LIN {X 0,Y 355.805,Z 517.624,A -85,B 0,C 180,E1 -17546.603,E2 -17546.603} C_VEL
LIN {X 0,Y 356.856,Z 517.924,A -85,B 0,C 180,E1 -17547.743,E2 -17547.743} C_VEL
LIN {X 0,Y 357.535,Z 518.046,A -85,B 0,C 180,E1 -17548.874,E2 -17548.874} C_VEL
LIN {X 0,Y 357.744,Z 518.094,A -85,B 0,C 180,E1 -17550,E2 -17550} C_VEL
LIN {X 0,Y 357.534,Z 518.031,A -85,B 0,C 180,E1 -17551.127,E2 -17551.127} C_VEL
LIN {X 0,Y 356.823,Z 517.932,A -85,B 0,C 180,E1 -17552.258,E2 -17552.258} C_VEL
LIN {X 0,Y 355.806,Z 517.611,A -85,B 0,C 180,E1 -17553.397,E2 -17553.397} C_VEL
LIN {X 0,Y 354.452,Z 517.067,A -85,B 0,C 180,E1 -17554.549,E2 -17554.549} C_VEL
LIN {X 0,Y 352.887,Z 516.184,A -85,B 0,C 180,E1 -17555.715,E2 -17555.715} C_VEL
LIN {X 0,Y 351.141,Z 514.881,A -85,B 0,C 180,E1 -17556.897,E2 -17556.897} C_VEL
LIN {X 0,Y 348.325,Z 512.278,A -85,B 0,C 180,E1 -17558.645,E2 -17558.645} C_VEL
LIN {X 0,Y 346.106,Z 510.135,A -85,B 0,C 180,E1 -17559.805,E2 -17559.805} C_VEL
LIN {X 0,Y 342.78,Z 507.679,A -85,B 0,C 180,E1 -17561.152,E2 -17561.152} C_VEL
LIN {X 0,Y 338.634,Z 503.933,A -85,B 0,C 180,E1 -17562.729,E2 -17562.729} C_VEL
LIN {X 0,Y 333.72,Z 499.517,A -85,B 0,C 180,E1 -17564.367,E2 -17564.367} C_VEL
LIN {X 0,Y 327.515,Z 493.449,A -85,B 0,C 180,E1 -17566.198,E2 -17566.198} C_VEL
LIN {X 0,Y 321.238,Z 487.195,A -85,B 0,C 180,E1 -17567.836,E2 -17567.836} C_VEL
LIN {X 0,Y 314.724,Z 480.337,A -85,B 0,C 180,E1 -17569.36,E2 -17569.36} C_VEL
LIN {X 0,Y 306.811,Z 471.536,A -85,B 0,C 180,E1 -17571.025,E2 -17571.025} C_VEL
LIN {X 0,Y 297.528,Z 460.121,A -85,B 0,C 180,E1 -17572.896,E2 -17572.896} C_VEL
LIN {X 0,Y 290.607,Z 450.33,A -85,B 0,C 180,E1 -17574.276,E2 -17574.276} C_VEL
LIN {X 0,Y 285.444,Z 441.391,A -85,B 0,C 180,E1 -17575.305,E2 -17575.305} C_VEL
LIN {X 0,Y 279.385,Z 428.404,A -85,B 0,C 180,E1 -17576.454,E2 -17576.454} C_VEL
LIN {X 0,Y 277.455,Z 424.082,A -85,B 0,C 180,E1 -17576.78,E2 -17576.78} C_VEL
LIN {X 0,Y 277.336,Z 423.44,A -85,B 0,C 180,E1 -17576.813,E2 -17576.813} C_VEL
LIN {X 0,Y 277.268,Z 423.449,A -85,B 0,C 180,E1 -17580.482,E2 -17580.482} C_VEL
LIN {X 0,Y 277.251,Z 423.449,A -85,B 0,C 180,E1 -17583.895,E2 -17583.895} C_VEL
LIN {X 0,Y 277.287,Z 423.444,A -85,B 0,C 180,E1 -17587.466,E2 -17587.466} C_VEL
LIN {X 0,Y 277.262,Z 423.447,A -85,B 0,C 180,E1 -17591.227,E2 -17591.227} C_VEL
LIN {X 0,Y 277.239,Z 423.449,A -85,B 0,C 180,E1 -17595.218,E2 -17595.218} C_VEL
LIN {X 0,Y 277.221,Z 423.451,A -85,B 0,C 180,E1 -17599.512,E2 -17599.512} C_VEL
LIN {X 0,Y 277.277,Z 423.446,A -85,B 0,C 180,E1 -17602.533,E2 -17602.533} C_VEL
LIN {X 0,Y 277.251,Z 423.451,A -85,B 0,C 180,E1 -17606.106,E2 -17606.106} C_VEL
LIN {X 0,Y 277.258,Z 423.447,A -85,B 0,C 180,E1 -17609.539,E2 -17609.539} C_VEL
LIN {X 0,Y 277.356,Z 423.434,A -85,B 0,C 180,E1 -17612.865,E2 -17612.865} C_VEL
LIN {X 0,Y 277.326,Z 423.44,A -85,B 0,C 180,E1 -17616.08,E2 -17616.08} C_VEL
LIN {X 0,Y 277.342,Z 423.434,A -85,B 0,C 180,E1 -17620.767,E2 -17620.767} C_VEL
LIN {X 0,Y 277.432,Z 423.422,A -85,B 0,C 180,E1 -17625.327,E2 -17625.327} C_VEL
LIN {X 0,Y 277.504,Z 423.416,A -85,B 0,C 180,E1 -17629.789,E2 -17629.789} C_VEL
LIN {X 0,Y 277.651,Z 423.398,A -85,B 0,C 180,E1 -17632.73,E2 -17632.73} C_VEL
LIN {X 0,Y 277.819,Z 423.364,A -85,B 0,C 180,E1 -17638.551,E2 -17638.551} C_VEL
LIN {X 0,Y 277.82,Z 423.376,A -85,B 0,C 180,E1 -17641.45,E2 -17641.45} C_VEL
LIN {X 0,Y 277.652,Z 423.4,A -85,B 0,C 180,E1 -17647.272,E2 -17647.272} C_VEL
LIN {X 0,Y 277.505,Z 423.416,A -85,B 0,C 180,E1 -17650.212,E2 -17650.212} C_VEL
LIN {X 0,Y 277.434,Z 423.425,A -85,B 0,C 180,E1 -17654.675,E2 -17654.675} C_VEL
LIN {X 0,Y 277.344,Z 423.44,A -85,B 0,C 180,E1 -17659.235,E2 -17659.235} C_VEL
LIN {X 0,Y 277.318,Z 423.44,A -85,B 0,C 180,E1 -17664.171,E2 -17664.171} C_VEL
LIN {X 0,Y 277.305,Z 423.441,A -85,B 0,C 180,E1 -17666.304,E2 -17666.304} C_VEL
LIN {X 0,Y 276.642,Z 423.529,A -85,B 0,C 180,E1 -17667.516,E2 -17667.516} C_VEL
LIN {X 0,Y 273.724,Z 423.892,A -85,B 0,C 180,E1 -17669.489,E2 -17669.489} C_VEL
LIN {X 0,Y 271.291,Z 424.409,A -85,B 0,C 180,E1 -17671.09,E2 -17671.09} C_VEL
LIN {X 0,Y 270.324,Z 424.94,A -85,B 0,C 180,E1 -17672.33,E2 -17672.33} C_VEL
LIN {X 0,Y 270.288,Z 425.147,A -85,B 0,C 180,E1 -17672.748,E2 -17672.748} C_VEL
LIN {X 0,Y 270.646,Z 427.318,A -85,B 0,C 180,E1 -17676.674,E2 -17676.674} C_VEL
LIN {X 0,Y 271.072,Z 430.164,A -85,B 0,C 180,E1 -17681.247,E2 -17681.247} C_VEL
LIN {X 0,Y 271.313,Z 432.313,A -85,B 0,C 180,E1 -17684.38,E2 -17684.38} C_VEL
LIN {X 0,Y 271.394,Z 434.753,A -85,B 0,C 180,E1 -17687.678,E2 -17687.678} C_VEL
LIN {X 0,Y 271.049,Z 437.477,A -85,B 0,C 180,E1 -17691.067,E2 -17691.067} C_VEL
LIN {X 0,Y 270.38,Z 440.968,A -85,B 0,C 180,E1 -17695.121,E2 -17695.121} C_VEL
LIN {X 0,Y 269.721,Z 444.717,A -85,B 0,C 180,E1 -17699.303,E2 -17699.303} C_VEL
LIN {X 0,Y 269.252,Z 447.838,A -85,B 0,C 180,E1 -17702.648,E2 -17702.648} C_VEL
LIN {X 0,Y 270.086,Z 451.047,A -85,B 0,C 180,E1 -17702.876,E2 -17702.876} C_VEL
LIN {X 0,Y 273.605,Z 464.4,A -85,B 0,C 180,E1 -17704.033,E2 -17704.033} C_VEL
LIN {X 0,Y 275.695,Z 474.898,A -85,B 0,C 180,E1 -17705.107,E2 -17705.107} C_VEL
LIN {X 0,Y 276.978,Z 485.03,A -85,B 0,C 180,E1 -17706.287,E2 -17706.287} C_VEL
LIN {X 0,Y 277.683,Z 494.384,A -85,B 0,C 180,E1 -17707.542,E2 -17707.542} C_VEL
LIN {X 0,Y 277.693,Z 499.477,A -85,B 0,C 180,E1 -17708.276,E2 -17708.276} C_VEL
LIN {X 0,Y 275.78,Z 509.625,A -85,B 0,C 180,E1 -17709.877,E2 -17709.877} C_VEL
LIN {X 0,Y 274.264,Z 517.761,A -85,B 0,C 180,E1 -17711.466,E2 -17711.466} C_VEL
LIN {X 0,Y 272.829,Z 524.973,A -85,B 0,C 180,E1 -17713.154,E2 -17713.154} C_VEL
LIN {X 0,Y 271.488,Z 531.513,A -85,B 0,C 180,E1 -17714.997,E2 -17714.997} C_VEL
LIN {X 0,Y 270.522,Z 536.015,A -85,B 0,C 180,E1 -17716.478,E2 -17716.478} C_VEL
LIN {X 0,Y 269.51,Z 541.512,A -85,B 0,C 180,E1 -17718.721,E2 -17718.721} C_VEL
LIN {X 0,Y 268.783,Z 545.842,A -85,B 0,C 180,E1 -17720.974,E2 -17720.974} C_VEL
LIN {X 0,Y 268.481,Z 548.213,A -85,B 0,C 180,E1 -17722.479,E2 -17722.479} C_VEL
LIN {X 0,Y 268.216,Z 550.778,A -85,B 0,C 180,E1 -17724.695,E2 -17724.695} C_VEL
LIN {X 0,Y 268.174,Z 552.47,A -85,B 0,C 180,E1 -17726.995,E2 -17726.995} C_VEL
LIN {X 0,Y 268.18,Z 553.061,A -85,B 0,C 180,E1 -17728.498,E2 -17728.498} C_VEL
LIN {X 0,Y 268.18,Z 553.061,A -85,B 0,C 180,E1 -17731.501,E2 -17731.501} C_VEL
LIN {X 0,Y 268.174,Z 552.47,A -85,B 0,C 180,E1 -17733.004,E2 -17733.004} C_VEL
LIN {X 0,Y 268.303,Z 550.017,A -85,B 0,C 180,E1 -17736.014,E2 -17736.014} C_VEL
LIN {X 0,Y 268.619,Z 547.062,A -85,B 0,C 180,E1 -17738.273,E2 -17738.273} C_VEL
LIN {X 0,Y 269.245,Z 543.069,A -85,B 0,C 180,E1 -17740.528,E2 -17740.528} C_VEL
LIN {X 0,Y 270.139,Z 537.934,A -85,B 0,C 180,E1 -17742.775,E2 -17742.775} C_VEL
LIN {X 0,Y 271.225,Z 532.67,A -85,B 0,C 180,E1 -17744.633,E2 -17744.633} C_VEL
LIN {X 0,Y 272.503,Z 526.351,A -85,B 0,C 180,E1 -17746.48,E2 -17746.48} C_VEL
LIN {X 0,Y 274.014,Z 519.292,A -85,B 0,C 180,E1 -17748.188,E2 -17748.188} C_VEL
LIN {X 0,Y 275.03,Z 513.468,A -85,B 0,C 180,E1 -17749.402,E2 -17749.402} C_VEL
LIN {X 0,Y 276.596,Z 505.288,A -85,B 0,C 180,E1 -17750.837,E2 -17750.837} C_VEL
LIN {X 0,Y 277.891,Z 498.129,A -85,B 0,C 180,E1 -17751.902,E2 -17751.902} C_VEL
LIN {X 0,Y 277.357,Z 488.828,A -85,B 0,C 180,E1 -17753.222,E2 -17753.222} C_VEL
LIN {X 0,Y 276.224,Z 478.64,A -85,B 0,C 180,E1 -17754.473,E2 -17754.473} C_VEL
LIN {X 0,Y 274.544,Z 468.766,A -85,B 0,C 180,E1 -17755.53,E2 -17755.53} C_VEL
LIN {X 0,Y 272.201,Z 458.808,A -85,B 0,C 180,E1 -17756.472,E2 -17756.472} C_VEL
LIN {X 0,Y 269.316,Z 448.595,A -85,B 0,C 180,E1 -17757.303,E2 -17757.303} C_VEL
LIN {X 0,Y 269.25,Z 447.839,A -85,B 0,C 180,E1 -17757.351,E2 -17757.351} C_VEL
LIN {X 0,Y 269.771,Z 444.07,A -85,B 0,C 180,E1 -17761.401,E2 -17761.401} C_VEL
LIN {X 0,Y 270.366,Z 440.938,A -85,B 0,C 180,E1 -17764.88,E2 -17764.88} C_VEL
LIN {X 0,Y 271.046,Z 437.457,A -85,B 0,C 180,E1 -17768.932,E2 -17768.932} C_VEL
LIN {X 0,Y 271.389,Z 434.743,A -85,B 0,C 180,E1 -17772.322,E2 -17772.322} C_VEL
LIN {X 0,Y 271.307,Z 432.301,A -85,B 0,C 180,E1 -17775.619,E2 -17775.619} C_VEL
LIN {X 0,Y 270.971,Z 429.623,A -85,B 0,C 180,E1 -17779.577,E2 -17779.577} C_VEL
LIN {X 0,Y 270.606,Z 427.143,A -85,B 0,C 180,E1 -17783.619,E2 -17783.619} C_VEL
LIN {X 0,Y 270.333,Z 425.32,A -85,B 0,C 180,E1 -17786.91,E2 -17786.91} C_VEL
LIN {X 0,Y 270.202,Z 424.328,A -85,B 0,C 180,E1 -17789.128,E2 -17789.128} C_VEL
LIN {X 0,Y 270.263,Z 424.321,A -85,B 0,C 180,E1 -17792.144,E2 -17792.144} C_VEL
LIN {X 0,Y 270.275,Z 424.321,A -85,B 0,C 180,E1 -17795.518,E2 -17795.518} C_VEL
LIN {X 0,Y 270.298,Z 424.318,A -85,B 0,C 180,E1 -17800.243,E2 -17800.243} C_VEL
LIN {X 0,Y 270.399,Z 424.303,A -85,B 0,C 180,E1 -17804.934,E2 -17804.934} C_VEL
LIN {X 0,Y 270.438,Z 424.296,A -85,B 0,C 180,E1 -17809.518,E2 -17809.518} C_VEL
LIN {X 0,Y 270.607,Z 424.279,A -85,B 0,C 180,E1 -17812.538,E2 -17812.538} C_VEL
LIN {X 0,Y 270.783,Z 424.253,A -85,B 0,C 180,E1 -17818.512,E2 -17818.512} C_VEL
LIN {X 0,Y 270.782,Z 424.24,A -85,B 0,C 180,E1 -17821.486,E2 -17821.486} C_VEL
LIN {X 0,Y 270.606,Z 424.275,A -85,B 0,C 180,E1 -17827.46,E2 -17827.46} C_VEL
LIN {X 0,Y 270.436,Z 424.298,A -85,B 0,C 180,E1 -17830.48,E2 -17830.48} C_VEL
LIN {X 0,Y 270.397,Z 424.297,A -85,B 0,C 180,E1 -17835.064,E2 -17835.064} C_VEL
LIN {X 0,Y 270.296,Z 424.314,A -85,B 0,C 180,E1 -17839.755,E2 -17839.755} C_VEL
LIN {X 0,Y 270.268,Z 424.314,A -85,B 0,C 180,E1 -17844.585,E2 -17844.585} C_VEL
LIN {X 0,Y 270.265,Z 424.322,A -85,B 0,C 180,E1 -17847.908,E2 -17847.908} C_VEL
LIN {X 0,Y 270.179,Z 424.329,A -85,B 0,C 180,E1 -17851.348,E2 -17851.348} C_VEL
LIN {X 0,Y 270.21,Z 424.325,A -85,B 0,C 180,E1 -17854.903,E2 -17854.903} C_VEL
LIN {X 0,Y 270.216,Z 424.324,A -85,B 0,C 180,E1 -17858.717,E2 -17858.717} C_VEL
LIN {X 0,Y 270.226,Z 424.322,A -85,B 0,C 180,E1 -17862.547,E2 -17862.547} C_VEL
LIN {X 0,Y 270.23,Z 424.322,A -85,B 0,C 180,E1 -17866.735,E2 -17866.735} C_VEL
LIN {X 0,Y 270.245,Z 424.323,A -85,B 0,C 180,E1 -17869.448,E2 -17869.448} C_VEL
LIN {X 0,Y 270.252,Z 424.323,A -85,B 0,C 180,E1 -17873.721,E2 -17873.721} C_VEL
LIN {X 0,Y 270.199,Z 424.328,A -85,B 0,C 180,E1 -17876.893,E2 -17876.893} C_VEL
LIN {X 0,Y 270.224,Z 424.324,A -85,B 0,C 180,E1 -17880.387,E2 -17880.387} C_VEL
LIN {X 0,Y 270.292,Z 424.316,A -85,B 0,C 180,E1 -17882.436,E2 -17882.436} C_VEL
LIN {X 0,Y 271.238,Z 427.034,A -85,B 0,C 180,E1 -17882.635,E2 -17882.635} C_VEL
LIN {X 0,Y 277.009,Z 439.136,A -85,B 0,C 180,E1 -17883.726,E2 -17883.726} C_VEL
LIN {X 0,Y 281.643,Z 449.005,A -85,B 0,C 180,E1 -17884.788,E2 -17884.788} C_VEL
LIN {X 0,Y 287.444,Z 458.206,A -85,B 0,C 180,E1 -17886.055,E2 -17886.055} C_VEL
LIN {X 0,Y 294.179,Z 467.421,A -85,B 0,C 180,E1 -17887.528,E2 -17887.528} C_VEL
LIN {X 0,Y 304.319,Z 479.414,A -85,B 0,C 180,E1 -17889.733,E2 -17889.733} C_VEL
LIN {X 0,Y 312.848,Z 488.67,A -85,B 0,C 180,E1 -17891.67,E2 -17891.67} C_VEL
LIN {X 0,Y 318.244,Z 494.216,A -85,B 0,C 180,E1 -17893.006,E2 -17893.006} C_VEL
LIN {X 0,Y 324.415,Z 500.118,A -85,B 0,C 180,E1 -17894.656,E2 -17894.656} C_VEL
LIN {X 0,Y 330.188,Z 505.543,A -85,B 0,C 180,E1 -17896.46,E2 -17896.46} C_VEL
LIN {X 0,Y 334.168,Z 509.334,A -85,B 0,C 180,E1 -17897.86,E2 -17897.86} C_VEL
LIN {X 0,Y 338.789,Z 513.066,A -85,B 0,C 180,E1 -17899.618,E2 -17899.618} C_VEL
LIN {X 0,Y 341.625,Z 515.391,A -85,B 0,C 180,E1 -17900.914,E2 -17900.914} C_VEL
LIN {X 0,Y 345.072,Z 518.684,A -85,B 0,C 180,E1 -17902.981,E2 -17902.981} C_VEL
LIN {X 0,Y 346.856,Z 520.059,A -85,B 0,C 180,E1 -17904.186,E2 -17904.186} C_VEL
LIN {X 0,Y 348.468,Z 521.018,A -85,B 0,C 180,E1 -17905.373,E2 -17905.373} C_VEL
LIN {X 0,Y 349.853,Z 521.619,A -85,B 0,C 180,E1 -17906.545,E2 -17906.545} C_VEL
LIN {X 0,Y 350.949,Z 521.964,A -85,B 0,C 180,E1 -17907.705,E2 -17907.705} C_VEL
LIN {X 0,Y 351.691,Z 522.116,A -85,B 0,C 180,E1 -17908.855,E2 -17908.855} C_VEL
LIN {X 0,Y 351.927,Z 522.169,A -85,B 0,C 180,E1 -17910,E2 -17910} C_VEL
LIN {X 0,Y 351.503,Z 522.091,A -85,B 0,C 180,E1 -17911.422,E2 -17911.422} C_VEL
LIN {X 0,Y 350.926,Z 521.964,A -85,B 0,C 180,E1 -17912.296,E2 -17912.296} C_VEL
LIN {X 0,Y 349.852,Z 521.61,A -85,B 0,C 180,E1 -17913.455,E2 -17913.455} C_VEL
LIN {X 0,Y 348.46,Z 521.034,A -85,B 0,C 180,E1 -17914.628,E2 -17914.628} C_VEL
LIN {X 0,Y 346.357,Z 519.728,A -85,B 0,C 180,E1 -17916.145,E2 -17916.145} C_VEL
LIN {X 0,Y 343.074,Z 516.885,A -85,B 0,C 180,E1 -17918.245,E2 -17918.245} C_VEL
LIN {X 0,Y 340.788,Z 514.63,A -85,B 0,C 180,E1 -17919.496,E2 -17919.496} C_VEL
LIN {X 0,Y 336.689,Z 511.512,A -85,B 0,C 180,E1 -17921.17,E2 -17921.17} C_VEL
LIN {X 0,Y 333.433,Z 508.537,A -85,B 0,C 180,E1 -17922.427,E2 -17922.427} C_VEL
LIN {X 0,Y 328.737,Z 504.298,A -85,B 0,C 180,E1 -17924.004,E2 -17924.004} C_VEL
LIN {X 0,Y 323.411,Z 499.102,A -85,B 0,C 180,E1 -17925.642,E2 -17925.642} C_VEL
LIN {X 0,Y 318.25,Z 494.227,A -85,B 0,C 180,E1 -17927,E2 -17927} C_VEL
LIN {X 0,Y 312.849,Z 488.679,A -85,B 0,C 180,E1 -17928.331,E2 -17928.331} C_VEL
LIN {X 0,Y 302.712,Z 477.5,A -85,B 0,C 180,E1 -17930.628,E2 -17930.628} C_VEL
LIN {X 0,Y 294.181,Z 467.415,A -85,B 0,C 180,E1 -17932.473,E2 -17932.473} C_VEL
LIN {X 0,Y 286.462,Z 456.866,A -85,B 0,C 180,E1 -17934.153,E2 -17934.153} C_VEL
LIN {X 0,Y 280.871,Z 447.401,A -85,B 0,C 180,E1 -17935.397,E2 -17935.397} C_VEL
LIN {X 0,Y 276.355,Z 437.594,A -85,B 0,C 180,E1 -17936.413,E2 -17936.413} C_VEL
LIN {X 0,Y 270.48,Z 425.259,A -85,B 0,C 180,E1 -17937.501,E2 -17937.501} C_VEL
LIN {X 0,Y 270.282,Z 424.318,A -85,B 0,C 180,E1 -17937.594,E2 -17937.594} C_VEL
LIN {X 0,Y 270.181,Z 424.329,A -85,B 0,C 180,E1 -17941.348,E2 -17941.348} C_VEL
LIN {X 0,Y 270.212,Z 424.327,A -85,B 0,C 180,E1 -17944.904,E2 -17944.904} C_VEL
LIN {X 0,Y 270.219,Z 424.326,A -85,B 0,C 180,E1 -17948.717,E2 -17948.717} C_VEL
LIN {X 0,Y 270.219,Z 424.326,A -85,B 0,C 180,E1 -17952.549,E2 -17952.549} C_VEL
LIN {X 0,Y 270.185,Z 424.328,A -85,B 0,C 180,E1 -17956.746,E2 -17956.746} C_VEL
LIN {X 0,Y 270.203,Z 424.325,A -85,B 0,C 180,E1 -17961.375,E2 -17961.375} C_VEL
LIN {X 0,Y 270.22,Z 424.323,A -85,B 0,C 180,E1 -17965.098,E2 -17965.098} C_VEL
LIN {X 0,Y 270.197,Z 424.326,A -85,B 0,C 180,E1 -17969.131,E2 -17969.131} C_VEL
LIN {X 0,Y 270.261,Z 424.322,A -85,B 0,C 180,E1 -17972.147,E2 -17972.147} C_VEL
LIN {X 0,Y 270.274,Z 424.313,A -85,B 0,C 180,E1 -17975.52,E2 -17975.52} C_VEL
LIN {X 0,Y 270.299,Z 424.313,A -85,B 0,C 180,E1 -17980.245,E2 -17980.245} C_VEL
LIN {X 0,Y 270.4,Z 424.297,A -85,B 0,C 180,E1 -17984.936,E2 -17984.936} C_VEL
LIN {X 0,Y 270.439,Z 424.297,A -85,B 0,C 180,E1 -17989.52,E2 -17989.52} C_VEL
LIN {X 0,Y 270.609,Z 424.275,A -85,B 0,C 180,E1 -17992.54,E2 -17992.54} C_VEL
LIN {X 0,Y 270.785,Z 424.239,A -85,B 0,C 180,E1 -17998.514,E2 -17998.514} C_VEL
LIN {X 0,Y 270.785,Z 424.252,A -85,B 0,C 180,E1 -18001.488,E2 -18001.488} C_VEL
LIN {X 0,Y 270.61,Z 424.279,A -85,B 0,C 180,E1 -18007.462,E2 -18007.462} C_VEL
LIN {X 0,Y 270.441,Z 424.296,A -85,B 0,C 180,E1 -18010.482,E2 -18010.482} C_VEL
LIN {X 0,Y 270.402,Z 424.303,A -85,B 0,C 180,E1 -18015.065,E2 -18015.065} C_VEL
LIN {X 0,Y 270.301,Z 424.315,A -85,B 0,C 180,E1 -18019.756,E2 -18019.756} C_VEL
LIN {X 0,Y 270.274,Z 424.319,A -85,B 0,C 180,E1 -18024.586,E2 -18024.586} C_VEL
LIN {X 0,Y 270.27,Z 424.32,A -85,B 0,C 180,E1 -18027.91,E2 -18027.91} C_VEL
LIN {X 0,Y 270.195,Z 424.428,A -85,B 0,C 180,E1 -18031.348,E2 -18031.348} C_VEL
LIN {X 0,Y 270.288,Z 425.147,A -85,B 0,C 180,E1 -18032.748,E2 -18032.748} C_VEL
LIN {X 0,Y 269.753,Z 425.906,A -85,B 0,C 180,E1 -18033.985,E2 -18033.985} C_VEL
LIN {X 0,Y 267.044,Z 427.473,A -85,B 0,C 180,E1 -18035.995,E2 -18035.995} C_VEL
LIN {X 0,Y 264.743,Z 428.786,A -85,B 0,C 180,E1 -18037.628,E2 -18037.628} C_VEL
LIN {X 0,Y 263.843,Z 429.689,A -85,B 0,C 180,E1 -18038.894,E2 -18038.894} C_VEL
LIN {X 0,Y 263.82,Z 429.959,A -85,B 0,C 180,E1 -18039.322,E2 -18039.322} C_VEL
LIN {X 0,Y 264.099,Z 431.534,A -85,B 0,C 180,E1 -18041.831,E2 -18041.831} C_VEL
LIN {X 0,Y 264.332,Z 434.311,A -85,B 0,C 180,E1 -18045.88,E2 -18045.88} C_VEL
LIN {X 0,Y 264.316,Z 436.143,A -85,B 0,C 180,E1 -18048.338,E2 -18048.338} C_VEL
LIN {X 0,Y 263.778,Z 439.258,A -85,B 0,C 180,E1 -18052.208,E2 -18052.208} C_VEL
LIN {X 0,Y 263.187,Z 442.329,A -85,B 0,C 180,E1 -18055.891,E2 -18055.891} C_VEL
LIN {X 0,Y 262.626,Z 445.456,A -85,B 0,C 180,E1 -18059.44,E2 -18059.44} C_VEL
LIN {X 0,Y 262.223,Z 447.643,A -85,B 0,C 180,E1 -18061.859,E2 -18061.859} C_VEL
LIN {X 0,Y 263.126,Z 450.954,A -85,B 0,C 180,E1 -18062.103,E2 -18062.103} C_VEL
LIN {X 0,Y 266.715,Z 464.224,A -85,B 0,C 180,E1 -18063.314,E2 -18063.314} C_VEL
LIN {X 0,Y 268.981,Z 475.669,A -85,B 0,C 180,E1 -18064.543,E2 -18064.543} C_VEL
LIN {X 0,Y 270.26,Z 485.569,A -85,B 0,C 180,E1 -18065.754,E2 -18065.754} C_VEL
LIN {X 0,Y 270.914,Z 495.182,A -85,B 0,C 180,E1 -18067.1,E2 -18067.1} C_VEL
LIN {X 0,Y 270.857,Z 500.526,A -85,B 0,C 180,E1 -18067.899,E2 -18067.899} C_VEL
LIN {X 0,Y 269.123,Z 509.414,A -85,B 0,C 180,E1 -18069.357,E2 -18069.357} C_VEL
LIN {X 0,Y 267.339,Z 518.322,A -85,B 0,C 180,E1 -18071.157,E2 -18071.157} C_VEL
LIN {X 0,Y 266.03,Z 524.761,A -85,B 0,C 180,E1 -18072.71,E2 -18072.71} C_VEL
LIN {X 0,Y 264.624,Z 531.301,A -85,B 0,C 180,E1 -18074.598,E2 -18074.598} C_VEL
LIN {X 0,Y 263.603,Z 535.803,A -85,B 0,C 180,E1 -18076.116,E2 -18076.116} C_VEL
LIN {X 0,Y 262.515,Z 541.3,A -85,B 0,C 180,E1 -18078.417,E2 -18078.417} C_VEL
LIN {X 0,Y 261.752,Z 545.63,A -85,B 0,C 180,E1 -18080.729,E2 -18080.729} C_VEL
LIN {X 0,Y 261.407,Z 548,A -85,B 0,C 180,E1 -18082.274,E2 -18082.274} C_VEL
LIN {X 0,Y 261.126,Z 550.735,A -85,B 0,C 180,E1 -18084.769,E2 -18084.769} C_VEL
LIN {X 0,Y 261.09,Z 552.258,A -85,B 0,C 180,E1 -18086.914,E2 -18086.914} C_VEL
LIN {X 0,Y 261.109,Z 552.85,A -85,B 0,C 180,E1 -18088.457,E2 -18088.457} C_VEL
LIN {X 0,Y 261.109,Z 552.851,A -85,B 0,C 180,E1 -18091.542,E2 -18091.542} C_VEL
LIN {X 0,Y 261.09,Z 552.259,A -85,B 0,C 180,E1 -18093.086,E2 -18093.086} C_VEL
LIN {X 0,Y 261.233,Z 549.805,A -85,B 0,C 180,E1 -18096.177,E2 -18096.177} C_VEL
LIN {X 0,Y 261.571,Z 546.85,A -85,B 0,C 180,E1 -18098.498,E2 -18098.498} C_VEL
LIN {X 0,Y 262.238,Z 542.857,A -85,B 0,C 180,E1 -18100.812,E2 -18100.812} C_VEL
LIN {X 0,Y 263.188,Z 537.722,A -85,B 0,C 180,E1 -18103.119,E2 -18103.119} C_VEL
LIN {X 0,Y 264.332,Z 532.458,A -85,B 0,C 180,E1 -18105.024,E2 -18105.024} C_VEL
LIN {X 0,Y 265.68,Z 526.139,A -85,B 0,C 180,E1 -18106.916,E2 -18106.916} C_VEL
LIN {X 0,Y 267.022,Z 520.188,A -85,B 0,C 180,E1 -18108.411,E2 -18108.411} C_VEL
LIN {X 0,Y 268.32,Z 513.256,A -85,B 0,C 180,E1 -18109.907,E2 -18109.907} C_VEL
LIN {X 0,Y 269.931,Z 505.076,A -85,B 0,C 180,E1 -18111.377,E2 -18111.377} C_VEL
LIN {X 0,Y 271.092,Z 499.27,A -85,B 0,C 180,E1 -18112.28,E2 -18112.28} C_VEL
LIN {X 0,Y 270.601,Z 489.407,A -85,B 0,C 180,E1 -18113.738,E2 -18113.738} C_VEL
LIN {X 0,Y 269.46,Z 478.85,A -85,B 0,C 180,E1 -18115.085,E2 -18115.085} C_VEL
LIN {X 0,Y 267.765,Z 468.955,A -85,B 0,C 180,E1 -18116.192,E2 -18116.192} C_VEL
LIN {X 0,Y 265.272,Z 458.49,A -85,B 0,C 180,E1 -18117.225,E2 -18117.225} C_VEL
LIN {X 0,Y 262.348,Z 448.706,A -85,B 0,C 180,E1 -18118.078,E2 -18118.078} C_VEL
LIN {X 0,Y 262.223,Z 447.612,A -85,B 0,C 180,E1 -18118.176,E2 -18118.176} C_VEL
LIN {X 0,Y 262.685,Z 444.949,A -85,B 0,C 180,E1 -18121.112,E2 -18121.112} C_VEL
LIN {X 0,Y 263.152,Z 442.304,A -85,B 0,C 180,E1 -18124.113,E2 -18124.113} C_VEL
LIN {X 0,Y 263.771,Z 439.175,A -85,B 0,C 180,E1 -18127.793,E2 -18127.793} C_VEL
LIN {X 0,Y 264.309,Z 436.115,A -85,B 0,C 180,E1 -18131.662,E2 -18131.662} C_VEL
LIN {X 0,Y 264.333,Z 434.309,A -85,B 0,C 180,E1 -18134.12,E2 -18134.12} C_VEL
LIN {X 0,Y 264.064,Z 431.455,A -85,B 0,C 180,E1 -18138.288,E2 -18138.288} C_VEL
LIN {X 0,Y 263.666,Z 429.049,A -85,B 0,C 180,E1 -18142.188,E2 -18142.188} C_VEL
LIN {X 0,Y 263.402,Z 426.948,A -85,B 0,C 180,E1 -18145.922,E2 -18145.922} C_VEL
LIN {X 0,Y 263.151,Z 425.206,A -85,B 0,C 180,E1 -18149.506,E2 -18149.506} C_VEL
LIN {X 0,Y 263.191,Z 425.205,A -85,B 0,C 180,E1 -18153.002,E2 -18153.002} C_VEL
LIN {X 0,Y 263.182,Z 425.206,A -85,B 0,C 180,E1 -18156.386,E2 -18156.386} C_VEL
LIN {X 0,Y 263.261,Z 425.193,A -85,B 0,C 180,E1 -18159.692,E2 -18159.692} C_VEL
LIN {X 0,Y 263.347,Z 425.183,A -85,B 0,C 180,E1 -18164.521,E2 -18164.521} C_VEL
LIN {X 0,Y 263.37,Z 425.177,A -85,B 0,C 180,E1 -18169.233,E2 -18169.233} C_VEL
LIN {X 0,Y 263.569,Z 425.155,A -85,B 0,C 180,E1 -18172.337,E2 -18172.337} C_VEL
LIN {X 0,Y 263.747,Z 425.129,A -85,B 0,C 180,E1 -18178.472,E2 -18178.472} C_VEL
LIN {X 0,Y 263.747,Z 425.115,A -85,B 0,C 180,E1 -18181.526,E2 -18181.526} C_VEL
LIN {X 0,Y 263.567,Z 425.153,A -85,B 0,C 180,E1 -18187.661,E2 -18187.661} C_VEL
LIN {X 0,Y 263.368,Z 425.177,A -85,B 0,C 180,E1 -18190.765,E2 -18190.765} C_VEL
LIN {X 0,Y 263.345,Z 425.176,A -85,B 0,C 180,E1 -18195.477,E2 -18195.477} C_VEL
LIN {X 0,Y 263.258,Z 425.19,A -85,B 0,C 180,E1 -18200.306,E2 -18200.306} C_VEL
LIN {X 0,Y 263.203,Z 425.193,A -85,B 0,C 180,E1 -18205.291,E2 -18205.291} C_VEL
LIN {X 0,Y 263.17,Z 425.201,A -85,B 0,C 180,E1 -18208.73,E2 -18208.73} C_VEL
LIN {X 0,Y 263.128,Z 425.208,A -85,B 0,C 180,E1 -18212.288,E2 -18212.288} C_VEL
LIN {X 0,Y 263.185,Z 425.202,A -85,B 0,C 180,E1 -18215.977,E2 -18215.977} C_VEL
LIN {X 0,Y 263.155,Z 425.206,A -85,B 0,C 180,E1 -18219.862,E2 -18219.862} C_VEL
LIN {X 0,Y 263.186,Z 425.202,A -85,B 0,C 180,E1 -18223.97,E2 -18223.97} C_VEL
LIN {X 0,Y 263.209,Z 425.198,A -85,B 0,C 180,E1 -18228.384,E2 -18228.384} C_VEL
LIN {X 0,Y 263.201,Z 425.201,A -85,B 0,C 180,E1 -18233.23,E2 -18233.23} C_VEL
LIN {X 0,Y 263.179,Z 425.203,A -85,B 0,C 180,E1 -18235.891,E2 -18235.891} C_VEL
LIN {X 0,Y 263.146,Z 425.208,A -85,B 0,C 180,E1 -18239.507,E2 -18239.507} C_VEL
LIN {X 0,Y 263.239,Z 425.356,A -85,B 0,C 180,E1 -18241.671,E2 -18241.671} C_VEL
LIN {X 0,Y 264.24,Z 428.061,A -85,B 0,C 180,E1 -18241.871,E2 -18241.871} C_VEL
LIN {X 0,Y 270.073,Z 439.995,A -85,B 0,C 180,E1 -18243.032,E2 -18243.032} C_VEL
LIN {X 0,Y 274.341,Z 449.708,A -85,B 0,C 180,E1 -18244.1,E2 -18244.1} C_VEL
LIN {X 0,Y 279.36,Z 458.841,A -85,B 0,C 180,E1 -18245.35,E2 -18245.35} C_VEL
LIN {X 0,Y 286.308,Z 468.777,A -85,B 0,C 180,E1 -18246.997,E2 -18246.997} C_VEL
LIN {X 0,Y 295.215,Z 479.692,A -85,B 0,C 180,E1 -18249.079,E2 -18249.079} C_VEL
LIN {X 0,Y 304.329,Z 489.654,A -85,B 0,C 180,E1 -18251.23,E2 -18251.23} C_VEL
LIN {X 0,Y 311.289,Z 496.914,A -85,B 0,C 180,E1 -18252.933,E2 -18252.933} C_VEL
LIN {X 0,Y 317.614,Z 503.043,A -85,B 0,C 180,E1 -18254.602,E2 -18254.602} C_VEL
LIN {X 0,Y 322.651,Z 507.913,A -85,B 0,C 180,E1 -18256.137,E2 -18256.137} C_VEL
LIN {X 0,Y 326.992,Z 511.865,A -85,B 0,C 180,E1 -18257.589,E2 -18257.589} C_VEL
LIN {X 0,Y 330.678,Z 515.161,A -85,B 0,C 180,E1 -18258.973,E2 -18258.973} C_VEL
LIN {X 0,Y 334.773,Z 518.27,A -85,B 0,C 180,E1 -18260.636,E2 -18260.636} C_VEL
LIN {X 0,Y 336.545,Z 519.984,A -85,B 0,C 180,E1 -18261.595,E2 -18261.595} C_VEL
LIN {X 0,Y 339.546,Z 522.728,A -85,B 0,C 180,E1 -18263.464,E2 -18263.464} C_VEL
LIN {X 0,Y 342.109,Z 524.43,A -85,B 0,C 180,E1 -18265.287,E2 -18265.287} C_VEL
LIN {X 0,Y 343.57,Z 525.106,A -85,B 0,C 180,E1 -18266.482,E2 -18266.482} C_VEL
LIN {X 0,Y 344.733,Z 525.526,A -85,B 0,C 180,E1 -18267.663,E2 -18267.663} C_VEL
LIN {X 0,Y 345.535,Z 525.727,A -85,B 0,C 180,E1 -18268.835,E2 -18268.835} C_VEL
LIN {X 0,Y 345.825,Z 525.776,A -85,B 0,C 180,E1 -18270,E2 -18270} C_VEL
LIN {X 0,Y 345.532,Z 525.715,A -85,B 0,C 180,E1 -18271.166,E2 -18271.166} C_VEL
LIN {X 0,Y 344.669,Z 525.505,A -85,B 0,C 180,E1 -18272.397,E2 -18272.397} C_VEL
LIN {X 0,Y 343.568,Z 525.105,A -85,B 0,C 180,E1 -18273.519,E2 -18273.519} C_VEL
LIN {X 0,Y 342.105,Z 524.449,A -85,B 0,C 180,E1 -18274.714,E2 -18274.714} C_VEL
LIN {X 0,Y 339.546,Z 522.749,A -85,B 0,C 180,E1 -18276.536,E2 -18276.536} C_VEL
LIN {X 0,Y 336.541,Z 520.012,A -85,B 0,C 180,E1 -18278.406,E2 -18278.406} C_VEL
LIN {X 0,Y 333.971,Z 517.673,A -85,B 0,C 180,E1 -18279.692,E2 -18279.692} C_VEL
LIN {X 0,Y 328.891,Z 513.6,A -85,B 0,C 180,E1 -18281.712,E2 -18281.712} C_VEL
LIN {X 0,Y 324.818,Z 509.797,A -85,B 0,C 180,E1 -18283.185,E2 -18283.185} C_VEL
LIN {X 0,Y 319.774,Z 505.182,A -85,B 0,C 180,E1 -18284.756,E2 -18284.756} C_VEL
LIN {X 0,Y 314.681,Z 500.242,A -85,B 0,C 180,E1 -18286.191,E2 -18286.191} C_VEL
LIN {X 0,Y 308.211,Z 493.741,A -85,B 0,C 180,E1 -18287.826,E2 -18287.826} C_VEL
LIN {X 0,Y 300.492,Z 485.615,A -85,B 0,C 180,E1 -18289.665,E2 -18289.665} C_VEL
LIN {X 0,Y 291.511,Z 475.332,A -85,B 0,C 180,E1 -18291.789,E2 -18291.789} C_VEL
LIN {X 0,Y 283.765,Z 465.367,A -85,B 0,C 180,E1 -18293.6,E2 -18293.6} C_VEL
LIN {X 0,Y 277.477,Z 455.646,A -85,B 0,C 180,E1 -18295.115,E2 -18295.115} C_VEL
LIN {X 0,Y 272.698,Z 446.227,A -85,B 0,C 180,E1 -18296.315,E2 -18296.315} C_VEL
LIN {X 0,Y 267.261,Z 433.941,A -85,B 0,C 180,E1 -18297.569,E2 -18297.569} C_VEL
LIN {X 0,Y 263.379,Z 426.063,A -85,B 0,C 180,E1 -18298.291,E2 -18298.291} C_VEL
LIN {X 0,Y 263.187,Z 425.203,A -85,B 0,C 180,E1 -18298.402,E2 -18298.402} C_VEL
LIN {X 0,Y 263.13,Z 425.21,A -85,B 0,C 180,E1 -18302.288,E2 -18302.288} C_VEL
LIN {X 0,Y 263.186,Z 425.202,A -85,B 0,C 180,E1 -18305.978,E2 -18305.978} C_VEL
LIN {X 0,Y 263.157,Z 425.205,A -85,B 0,C 180,E1 -18309.863,E2 -18309.863} C_VEL
LIN {X 0,Y 263.141,Z 425.207,A -85,B 0,C 180,E1 -18313.98,E2 -18313.98} C_VEL
LIN {X 0,Y 263.126,Z 425.21,A -85,B 0,C 180,E1 -18318.406,E2 -18318.406} C_VEL
LIN {X 0,Y 263.162,Z 425.205,A -85,B 0,C 180,E1 -18322.105,E2 -18322.105} C_VEL
LIN {X 0,Y 263.181,Z 425.203,A -85,B 0,C 180,E1 -18325.891,E2 -18325.891} C_VEL
LIN {X 0,Y 263.145,Z 425.205,A -85,B 0,C 180,E1 -18329.507,E2 -18329.507} C_VEL
LIN {X 0,Y 263.189,Z 425.199,A -85,B 0,C 180,E1 -18333.003,E2 -18333.003} C_VEL
LIN {X 0,Y 263.181,Z 425.202,A -85,B 0,C 180,E1 -18336.388,E2 -18336.388} C_VEL
LIN {X 0,Y 263.261,Z 425.19,A -85,B 0,C 180,E1 -18339.694,E2 -18339.694} C_VEL
LIN {X 0,Y 263.348,Z 425.176,A -85,B 0,C 180,E1 -18344.523,E2 -18344.523} C_VEL
LIN {X 0,Y 263.371,Z 425.177,A -85,B 0,C 180,E1 -18349.235,E2 -18349.235} C_VEL
LIN {X 0,Y 263.57,Z 425.152,A -85,B 0,C 180,E1 -18352.339,E2 -18352.339} C_VEL
LIN {X 0,Y 263.75,Z 425.115,A -85,B 0,C 180,E1 -18358.474,E2 -18358.474} C_VEL
LIN {X 0,Y 263.75,Z 425.129,A -85,B 0,C 180,E1 -18361.528,E2 -18361.528} C_VEL
LIN {X 0,Y 263.572,Z 425.155,A -85,B 0,C 180,E1 -18367.662,E2 -18367.662} C_VEL
LIN {X 0,Y 263.373,Z 425.177,A -85,B 0,C 180,E1 -18370.766,E2 -18370.766} C_VEL
LIN {X 0,Y 263.35,Z 425.183,A -85,B 0,C 180,E1 -18375.479,E2 -18375.479} C_VEL
LIN {X 0,Y 263.263,Z 425.191,A -85,B 0,C 180,E1 -18380.307,E2 -18380.307} C_VEL
LIN {X 0,Y 263.208,Z 425.201,A -85,B 0,C 180,E1 -18385.292,E2 -18385.292} C_VEL
LIN {X 0,Y 263.166,Z 425.207,A -85,B 0,C 180,E1 -18388.732,E2 -18388.732} C_VEL
LIN {X 0,Y 263.143,Z 425.21,A -85,B 0,C 180,E1 -18390.495,E2 -18390.495} C_VEL
LIN {X 0,Y 263.396,Z 427.016,A -85,B 0,C 180,E1 -18394.194,E2 -18394.194} C_VEL
LIN {X 0,Y 263.691,Z 429.046,A -85,B 0,C 180,E1 -18397.808,E2 -18397.808} C_VEL
LIN {X 0,Y 263.82,Z 429.959,A -85,B 0,C 180,E1 -18399.322,E2 -18399.322} C_VEL
LIN {X 0,Y 263.318,Z 430.832,A -85,B 0,C 180,E1 -18400.584,E2 -18400.584} C_VEL
LIN {X 0,Y 260.642,Z 432.557,A -85,B 0,C 180,E1 -18402.636,E2 -18402.636} C_VEL
LIN {X 0,Y 258.298,Z 434.005,A -85,B 0,C 180,E1 -18404.303,E2 -18404.303} C_VEL
LIN {X 0,Y 257.3,Z 435.031,A -85,B 0,C 180,E1 -18405.595,E2 -18405.595} C_VEL
LIN {X 0,Y 257.228,Z 435.347,A -85,B 0,C 180,E1 -18406.033,E2 -18406.033} C_VEL
LIN {X 0,Y 257.166,Z 437.531,A -85,B 0,C 180,E1 -18409.013,E2 -18409.013} C_VEL
LIN {X 0,Y 256.609,Z 440.613,A -85,B 0,C 180,E1 -18412.949,E2 -18412.949} C_VEL
LIN {X 0,Y 255.92,Z 443.716,A -85,B 0,C 180,E1 -18416.686,E2 -18416.686} C_VEL
LIN {X 0,Y 255.267,Z 447.441,A -85,B 0,C 180,E1 -18421.023,E2 -18421.023} C_VEL
LIN {X 0,Y 256.12,Z 450.668,A -85,B 0,C 180,E1 -18421.268,E2 -18421.268} C_VEL
LIN {X 0,Y 259.671,Z 463.203,A -85,B 0,C 180,E1 -18422.464,E2 -18422.464} C_VEL
LIN {X 0,Y 261.952,Z 474.325,A -85,B 0,C 180,E1 -18423.691,E2 -18423.691} C_VEL
LIN {X 0,Y 263.348,Z 484.09,A -85,B 0,C 180,E1 -18424.914,E2 -18424.914} C_VEL
LIN {X 0,Y 264.052,Z 493.375,A -85,B 0,C 180,E1 -18426.227,E2 -18426.227} C_VEL
LIN {X 0,Y 264.27,Z 500.314,A -85,B 0,C 180,E1 -18427.318,E2 -18427.318} C_VEL
LIN {X 0,Y 262.463,Z 509.202,A -85,B 0,C 180,E1 -18428.808,E2 -18428.808} C_VEL
LIN {X 0,Y 260.654,Z 517.801,A -85,B 0,C 180,E1 -18430.577,E2 -18430.577} C_VEL
LIN {X 0,Y 259.254,Z 524.55,A -85,B 0,C 180,E1 -18432.243,E2 -18432.243} C_VEL
LIN {X 0,Y 257.759,Z 531.089,A -85,B 0,C 180,E1 -18434.177,E2 -18434.177} C_VEL
LIN {X 0,Y 256.704,Z 535.591,A -85,B 0,C 180,E1 -18435.735,E2 -18435.735} C_VEL
LIN {X 0,Y 255.532,Z 541.087,A -85,B 0,C 180,E1 -18438.096,E2 -18438.096} C_VEL
LIN {X 0,Y 254.739,Z 545.418,A -85,B 0,C 180,E1 -18440.472,E2 -18440.472} C_VEL
LIN {X 0,Y 254.355,Z 547.788,A -85,B 0,C 180,E1 -18442.059,E2 -18442.059} C_VEL
LIN {X 0,Y 254.024,Z 550.716,A -85,B 0,C 180,E1 -18444.881,E2 -18444.881} C_VEL
LIN {X 0,Y 253.988,Z 552.047,A -85,B 0,C 180,E1 -18446.827,E2 -18446.827} C_VEL
LIN {X 0,Y 254.016,Z 552.639,A -85,B 0,C 180,E1 -18448.414,E2 -18448.414} C_VEL
LIN {X 0,Y 254.016,Z 552.64,A -85,B 0,C 180,E1 -18451.585,E2 -18451.585} C_VEL
LIN {X 0,Y 253.988,Z 552.047,A -85,B 0,C 180,E1 -18453.172,E2 -18453.172} C_VEL
LIN {X 0,Y 254.162,Z 549.593,A -85,B 0,C 180,E1 -18456.35,E2 -18456.35} C_VEL
LIN {X 0,Y 254.52,Z 546.637,A -85,B 0,C 180,E1 -18458.735,E2 -18458.735} C_VEL
LIN {X 0,Y 255.221,Z 542.644,A -85,B 0,C 180,E1 -18461.113,E2 -18461.113} C_VEL
LIN {X 0,Y 256.256,Z 537.51,A -85,B 0,C 180,E1 -18463.48,E2 -18463.48} C_VEL
LIN {X 0,Y 257.463,Z 532.246,A -85,B 0,C 180,E1 -18465.435,E2 -18465.435} C_VEL
LIN {X 0,Y 258.882,Z 525.927,A -85,B 0,C 180,E1 -18467.374,E2 -18467.374} C_VEL
LIN {X 0,Y 260.225,Z 519.975,A -85,B 0,C 180,E1 -18468.91,E2 -18468.91} C_VEL
LIN {X 0,Y 261.633,Z 513.044,A -85,B 0,C 180,E1 -18470.438,E2 -18470.438} C_VEL
LIN {X 0,Y 263.315,Z 504.864,A -85,B 0,C 180,E1 -18471.941,E2 -18471.941} C_VEL
LIN {X 0,Y 264.345,Z 499.052,A -85,B 0,C 180,E1 -18472.881,E2 -18472.881} C_VEL
LIN {X 0,Y 263.799,Z 489.242,A -85,B 0,C 180,E1 -18474.383,E2 -18474.383} C_VEL
LIN {X 0,Y 262.727,Z 479.113,A -85,B 0,C 180,E1 -18475.723,E2 -18475.723} C_VEL
LIN {X 0,Y 260.782,Z 468.161,A -85,B 0,C 180,E1 -18476.996,E2 -18476.996} C_VEL
LIN {X 0,Y 258.246,Z 457.755,A -85,B 0,C 180,E1 -18478.061,E2 -18478.061} C_VEL
LIN {X 0,Y 255.342,Z 448.214,A -85,B 0,C 180,E1 -18478.93,E2 -18478.93} C_VEL
LIN {X 0,Y 255.264,Z 447.444,A -85,B 0,C 180,E1 -18478.976,E2 -18478.976} C_VEL
LIN {X 0,Y 255.895,Z 443.655,A -85,B 0,C 180,E1 -18483.317,E2 -18483.317} C_VEL
LIN {X 0,Y 256.664,Z 440.26,A -85,B 0,C 180,E1 -18487.43,E2 -18487.43} C_VEL
LIN {X 0,Y 257.16,Z 437.49,A -85,B 0,C 180,E1 -18490.987,E2 -18490.987} C_VEL
LIN {X 0,Y 257.274,Z 435.947,A -85,B 0,C 180,E1 -18493.072,E2 -18493.072} C_VEL
LIN {X 0,Y 257.108,Z 433.344,A -85,B 0,C 180,E1 -18496.891,E2 -18496.891} C_VEL
LIN {X 0,Y 256.74,Z 430.794,A -85,B 0,C 180,E1 -18500.978,E2 -18500.978} C_VEL
LIN {X 0,Y 256.398,Z 428.363,A -85,B 0,C 180,E1 -18505.315,E2 -18505.315} C_VEL
LIN {X 0,Y 256.177,Z 426.712,A -85,B 0,C 180,E1 -18508.583,E2 -18508.583} C_VEL
LIN {X 0,Y 256.113,Z 426.084,A -85,B 0,C 180,E1 -18510.399,E2 -18510.399} C_VEL
LIN {X 0,Y 256.186,Z 426.079,A -85,B 0,C 180,E1 -18514.86,E2 -18514.86} C_VEL
LIN {X 0,Y 256.164,Z 426.079,A -85,B 0,C 180,E1 -18519.104,E2 -18519.104} C_VEL
LIN {X 0,Y 256.297,Z 426.059,A -85,B 0,C 180,E1 -18524.084,E2 -18524.084} C_VEL
LIN {X 0,Y 256.306,Z 426.059,A -85,B 0,C 180,E1 -18528.933,E2 -18528.933} C_VEL
LIN {X 0,Y 256.536,Z 426.03,A -85,B 0,C 180,E1 -18532.126,E2 -18532.126} C_VEL
LIN {X 0,Y 256.71,Z 426.006,A -85,B 0,C 180,E1 -18538.43,E2 -18538.43} C_VEL
LIN {X 0,Y 256.71,Z 425.99,A -85,B 0,C 180,E1 -18541.568,E2 -18541.568} C_VEL
LIN {X 0,Y 256.535,Z 426.03,A -85,B 0,C 180,E1 -18547.872,E2 -18547.872} C_VEL
LIN {X 0,Y 256.304,Z 426.056,A -85,B 0,C 180,E1 -18551.065,E2 -18551.065} C_VEL
LIN {X 0,Y 256.294,Z 426.056,A -85,B 0,C 180,E1 -18555.914,E2 -18555.914} C_VEL
LIN {X 0,Y 256.161,Z 426.073,A -85,B 0,C 180,E1 -18560.895,E2 -18560.895} C_VEL
LIN {X 0,Y 256.183,Z 426.067,A -85,B 0,C 180,E1 -18565.138,E2 -18565.138} C_VEL
LIN {X 0,Y 256.106,Z 426.083,A -85,B 0,C 180,E1 -18569.6,E2 -18569.6} C_VEL
LIN {X 0,Y 256.08,Z 426.086,A -85,B 0,C 180,E1 -18573.29,E2 -18573.29} C_VEL
LIN {X 0,Y 256.136,Z 426.079,A -85,B 0,C 180,E1 -18577.279,E2 -18577.279} C_VEL
LIN {X 0,Y 256.117,Z 426.08,A -85,B 0,C 180,E1 -18581.19,E2 -18581.19} C_VEL
LIN {X 0,Y 256.112,Z 426.081,A -85,B 0,C 180,E1 -18584.483,E2 -18584.483} C_VEL
LIN {X 0,Y 256.129,Z 426.079,A -85,B 0,C 180,E1 -18588.812,E2 -18588.812} C_VEL
LIN {X 0,Y 256.15,Z 426.077,A -85,B 0,C 180,E1 -18592.872,E2 -18592.872} C_VEL
LIN {X 0,Y 256.08,Z 426.086,A -85,B 0,C 180,E1 -18596.71,E2 -18596.71} C_VEL
LIN {X 0,Y 256.108,Z 426.088,A -85,B 0,C 180,E1 -18600.823,E2 -18600.823} C_VEL
LIN {X 0,Y 257.057,Z 428.839,A -85,B 0,C 180,E1 -18601.029,E2 -18601.029} C_VEL
LIN {X 0,Y 262.273,Z 439.021,A -85,B 0,C 180,E1 -18602.095,E2 -18602.095} C_VEL
LIN {X 0,Y 267.381,Z 451.07,A -85,B 0,C 180,E1 -18603.46,E2 -18603.46} C_VEL
LIN {X 0,Y 272.005,Z 460.071,A -85,B 0,C 180,E1 -18604.73,E2 -18604.73} C_VEL
LIN {X 0,Y 277.99,Z 469.509,A -85,B 0,C 180,E1 -18606.32,E2 -18606.32} C_VEL
LIN {X 0,Y 286.908,Z 480.795,A -85,B 0,C 180,E1 -18608.563,E2 -18608.563} C_VEL
LIN {X 0,Y 295.801,Z 490.732,A -85,B 0,C 180,E1 -18610.807,E2 -18610.807} C_VEL
LIN {X 0,Y 304.842,Z 499.936,A -85,B 0,C 180,E1 -18613.087,E2 -18613.087} C_VEL
LIN {X 0,Y 311.309,Z 506.191,A -85,B 0,C 180,E1 -18614.816,E2 -18614.816} C_VEL
LIN {X 0,Y 316.781,Z 511.403,A -85,B 0,C 180,E1 -18616.477,E2 -18616.477} C_VEL
LIN {X 0,Y 321.342,Z 515.623,A -85,B 0,C 180,E1 -18618.009,E2 -18618.009} C_VEL
LIN {X 0,Y 325.023,Z 518.794,A -85,B 0,C 180,E1 -18619.409,E2 -18619.409} C_VEL
LIN {X 0,Y 327.778,Z 520.887,A -85,B 0,C 180,E1 -18620.501,E2 -18620.501} C_VEL
LIN {X 0,Y 330.784,Z 523.66,A -85,B 0,C 180,E1 -18622.062,E2 -18622.062} C_VEL
LIN {X 0,Y 333.717,Z 526.195,A -85,B 0,C 180,E1 -18623.956,E2 -18623.956} C_VEL
LIN {X 0,Y 335.441,Z 527.314,A -85,B 0,C 180,E1 -18625.193,E2 -18625.193} C_VEL
LIN {X 0,Y 337.76,Z 528.435,A -85,B 0,C 180,E1 -18627.139,E2 -18627.139} C_VEL
LIN {X 0,Y 339.117,Z 528.845,A -85,B 0,C 180,E1 -18628.813,E2 -18628.813} C_VEL
LIN {X 0,Y 339.463,Z 528.905,A -85,B 0,C 180,E1 -18630,E2 -18630} C_VEL
LIN {X 0,Y 339.112,Z 528.835,A -85,B 0,C 180,E1 -18631.188,E2 -18631.188} C_VEL
LIN {X 0,Y 337.76,Z 528.445,A -85,B 0,C 180,E1 -18632.862,E2 -18632.862} C_VEL
LIN {X 0,Y 335.439,Z 527.336,A -85,B 0,C 180,E1 -18634.808,E2 -18634.808} C_VEL
LIN {X 0,Y 332.626,Z 525.357,A -85,B 0,C 180,E1 -18636.763,E2 -18636.763} C_VEL
LIN {X 0,Y 329.624,Z 522.554,A -85,B 0,C 180,E1 -18638.584,E2 -18638.584} C_VEL
LIN {X 0,Y 326.718,Z 520.099,A -85,B 0,C 180,E1 -18639.909,E2 -18639.909} C_VEL
LIN {X 0,Y 322.708,Z 516.829,A -85,B 0,C 180,E1 -18641.477,E2 -18641.477} C_VEL
LIN {X 0,Y 317.683,Z 512.238,A -85,B 0,C 180,E1 -18643.249,E2 -18643.249} C_VEL
LIN {X 0,Y 311.322,Z 506.136,A -85,B 0,C 180,E1 -18645.193,E2 -18645.193} C_VEL
LIN {X 0,Y 303.56,Z 498.589,A -85,B 0,C 180,E1 -18647.254,E2 -18647.254} C_VEL
LIN {X 0,Y 293.158,Z 487.902,A -85,B 0,C 180,E1 -18649.87,E2 -18649.87} C_VEL
LIN {X 0,Y 283.518,Z 476.796,A -85,B 0,C 180,E1 -18652.275,E2 -18652.275} C_VEL
LIN {X 0,Y 276.908,Z 467.78,A -85,B 0,C 180,E1 -18653.982,E2 -18653.982} C_VEL
LIN {X 0,Y 271.511,Z 459.299,A -85,B 0,C 180,E1 -18655.394,E2 -18655.394} C_VEL
LIN {X 0,Y 267.217,Z 450.638,A -85,B 0,C 180,E1 -18656.593,E2 -18656.593} C_VEL
LIN {X 0,Y 261.538,Z 437.482,A -85,B 0,C 180,E1 -18658.068,E2 -18658.068} C_VEL
LIN {X 0,Y 256.381,Z 427.346,A -85,B 0,C 180,E1 -18659.103,E2 -18659.103} C_VEL
LIN {X 0,Y 256.122,Z 426.082,A -85,B 0,C 180,E1 -18659.206,E2 -18659.206} C_VEL
LIN {X 0,Y 256.082,Z 426.086,A -85,B 0,C 180,E1 -18663.291,E2 -18663.291} C_VEL
LIN {X 0,Y 256.138,Z 426.079,A -85,B 0,C 180,E1 -18667.279,E2 -18667.279} C_VEL
LIN {X 0,Y 256.101,Z 426.083,A -85,B 0,C 180,E1 -18671.194,E2 -18671.194} C_VEL
LIN {X 0,Y 256.069,Z 426.086,A -85,B 0,C 180,E1 -18675.527,E2 -18675.527} C_VEL
LIN {X 0,Y 256.057,Z 426.088,A -85,B 0,C 180,E1 -18678.798,E2 -18678.798} C_VEL
LIN {X 0,Y 256.141,Z 426.078,A -85,B 0,C 180,E1 -18682.87,E2 -18682.87} C_VEL
LIN {X 0,Y 256.082,Z 426.085,A -85,B 0,C 180,E1 -18686.711,E2 -18686.711} C_VEL
LIN {X 0,Y 256.132,Z 426.078,A -85,B 0,C 180,E1 -18691.407,E2 -18691.407} C_VEL
LIN {X 0,Y 256.164,Z 426.072,A -85,B 0,C 180,E1 -18695.7,E2 -18695.7} C_VEL
LIN {X 0,Y 256.164,Z 426.073,A -85,B 0,C 180,E1 -18699.106,E2 -18699.106} C_VEL
LIN {X 0,Y 256.297,Z 426.056,A -85,B 0,C 180,E1 -18704.086,E2 -18704.086} C_VEL
LIN {X 0,Y 256.307,Z 426.056,A -85,B 0,C 180,E1 -18708.935,E2 -18708.935} C_VEL
LIN {X 0,Y 256.538,Z 426.03,A -85,B 0,C 180,E1 -18712.128,E2 -18712.128} C_VEL
LIN {X 0,Y 256.713,Z 425.99,A -85,B 0,C 180,E1 -18718.432,E2 -18718.432} C_VEL
LIN {X 0,Y 256.713,Z 426.005,A -85,B 0,C 180,E1 -18721.57,E2 -18721.57} C_VEL
LIN {X 0,Y 256.539,Z 426.029,A -85,B 0,C 180,E1 -18727.874,E2 -18727.874} C_VEL
LIN {X 0,Y 256.309,Z 426.059,A -85,B 0,C 180,E1 -18731.067,E2 -18731.067} C_VEL
LIN {X 0,Y 256.299,Z 426.059,A -85,B 0,C 180,E1 -18735.916,E2 -18735.916} C_VEL
LIN {X 0,Y 256.167,Z 426.077,A -85,B 0,C 180,E1 -18740.896,E2 -18740.896} C_VEL
LIN {X 0,Y 256.188,Z 426.075,A -85,B 0,C 180,E1 -18745.139,E2 -18745.139} C_VEL
LIN {X 0,Y 256.105,Z 426.087,A -85,B 0,C 180,E1 -18749.602,E2 -18749.602} C_VEL
LIN {X 0,Y 256.289,Z 427.629,A -85,B 0,C 180,E1 -18753.261,E2 -18753.261} C_VEL
LIN {X 0,Y 256.636,Z 429.878,A -85,B 0,C 180,E1 -18757.424,E2 -18757.424} C_VEL
LIN {X 0,Y 256.958,Z 432.017,A -85,B 0,C 180,E1 -18761.028,E2 -18761.028} C_VEL
LIN {X 0,Y 257.211,Z 434.443,A -85,B 0,C 180,E1 -18764.731,E2 -18764.731} C_VEL
LIN {X 0,Y 257.228,Z 435.347,A -85,B 0,C 180,E1 -18766.033,E2 -18766.033} C_VEL
LIN {X 0,Y 256.555,Z 436.358,A -85,B 0,C 180,E1 -18767.319,E2 -18767.319} C_VEL
LIN {X 0,Y 254.911,Z 437.491,A -85,B 0,C 180,E1 -18768.573,E2 -18768.573} C_VEL
LIN {X 0,Y 250.916,Z 439.81,A -85,B 0,C 180,E1 -18771.087,E2 -18771.087} C_VEL
LIN {X 0,Y 249.669,Z 440.929,A -85,B 0,C 180,E1 -18772.404,E2 -18772.404} C_VEL
LIN {X 0,Y 249.509,Z 441.288,A -85,B 0,C 180,E1 -18772.854,E2 -18772.854} C_VEL
LIN {X 0,Y 249.048,Z 443.538,A -85,B 0,C 180,E1 -18775.64,E2 -18775.64} C_VEL
LIN {X 0,Y 248.313,Z 447.305,A -85,B 0,C 180,E1 -18780.14,E2 -18780.14} C_VEL
LIN {X 0,Y 249.218,Z 450.563,A -85,B 0,C 180,E1 -18780.4,E2 -18780.4} C_VEL
LIN {X 0,Y 252.952,Z 463.645,A -85,B 0,C 180,E1 -18781.726,E2 -18781.726} C_VEL
LIN {X 0,Y 255.058,Z 473.712,A -85,B 0,C 180,E1 -18782.881,E2 -18782.881} C_VEL
LIN {X 0,Y 256.628,Z 484.419,A -85,B 0,C 180,E1 -18784.283,E2 -18784.283} C_VEL
LIN {X 0,Y 257.265,Z 493.382,A -85,B 0,C 180,E1 -18785.595,E2 -18785.595} C_VEL
LIN {X 0,Y 257.47,Z 501.245,A -85,B 0,C 180,E1 -18786.897,E2 -18786.897} C_VEL
LIN {X 0,Y 255.807,Z 508.989,A -85,B 0,C 180,E1 -18788.229,E2 -18788.229} C_VEL
LIN {X 0,Y 254.176,Z 516.505,A -85,B 0,C 180,E1 -18789.781,E2 -18789.781} C_VEL
LIN {X 0,Y 252.48,Z 524.402,A -85,B 0,C 180,E1 -18791.77,E2 -18791.77} C_VEL
LIN {X 0,Y 250.901,Z 530.877,A -85,B 0,C 180,E1 -18793.733,E2 -18793.733} C_VEL
LIN {X 0,Y 249.82,Z 535.38,A -85,B 0,C 180,E1 -18795.334,E2 -18795.334} C_VEL
LIN {X 0,Y 248.562,Z 540.875,A -85,B 0,C 180,E1 -18797.757,E2 -18797.757} C_VEL
LIN {X 0,Y 247.703,Z 545.206,A -85,B 0,C 180,E1 -18800.198,E2 -18800.198} C_VEL
LIN {X 0,Y 247.299,Z 547.576,A -85,B 0,C 180,E1 -18801.831,E2 -18801.831} C_VEL
LIN {X 0,Y 246.947,Z 550.652,A -85,B 0,C 180,E1 -18804.936,E2 -18804.936} C_VEL
LIN {X 0,Y 246.89,Z 551.835,A -85,B 0,C 180,E1 -18806.736,E2 -18806.736} C_VEL
LIN {X 0,Y 246.925,Z 552.428,A -85,B 0,C 180,E1 -18808.369,E2 -18808.369} C_VEL
LIN {X 0,Y 246.957,Z 552.584,A -85,B 0,C 180,E1 -18810,E2 -18810} C_VEL
LIN {X 0,Y 246.925,Z 552.428,A -85,B 0,C 180,E1 -18811.631,E2 -18811.631} C_VEL
LIN {X 0,Y 246.891,Z 551.835,A -85,B 0,C 180,E1 -18813.263,E2 -18813.263} C_VEL
LIN {X 0,Y 247.075,Z 549.381,A -85,B 0,C 180,E1 -18816.533,E2 -18816.533} C_VEL
LIN {X 0,Y 247.491,Z 546.426,A -85,B 0,C 180,E1 -18818.985,E2 -18818.985} C_VEL
LIN {X 0,Y 248.224,Z 542.432,A -85,B 0,C 180,E1 -18821.431,E2 -18821.431} C_VEL
LIN {X 0,Y 249.314,Z 537.297,A -85,B 0,C 180,E1 -18823.863,E2 -18823.863} C_VEL
LIN {X 0,Y 250.609,Z 532.034,A -85,B 0,C 180,E1 -18825.868,E2 -18825.868} C_VEL
LIN {X 0,Y 252.109,Z 525.715,A -85,B 0,C 180,E1 -18827.857,E2 -18827.857} C_VEL
LIN {X 0,Y 253.572,Z 519.284,A -85,B 0,C 180,E1 -18829.549,E2 -18829.549} C_VEL
LIN {X 0,Y 254.958,Z 512.832,A -85,B 0,C 180,E1 -18830.998,E2 -18830.998} C_VEL
LIN {X 0,Y 256.734,Z 504.652,A -85,B 0,C 180,E1 -18832.534,E2 -18832.534} C_VEL
LIN {X 0,Y 257.577,Z 500.102,A -85,B 0,C 180,E1 -18833.305,E2 -18833.305} C_VEL
LIN {X 0,Y 256.968,Z 488.272,A -85,B 0,C 180,E1 -18835.173,E2 -18835.173} C_VEL
LIN {X 0,Y 255.788,Z 478.308,A -85,B 0,C 180,E1 -18836.537,E2 -18836.537} C_VEL
LIN {X 0,Y 254.044,Z 468.613,A -85,B 0,C 180,E1 -18837.714,E2 -18837.714} C_VEL
LIN {X 0,Y 251.756,Z 459.154,A -85,B 0,C 180,E1 -18838.746,E2 -18838.746} C_VEL
LIN {X 0,Y 248.381,Z 447.923,A -85,B 0,C 180,E1 -18839.824,E2 -18839.824} C_VEL
LIN {X 0,Y 248.306,Z 447.229,A -85,B 0,C 180,E1 -18839.882,E2 -18839.882} C_VEL
LIN {X 0,Y 249.03,Z 443.444,A -85,B 0,C 180,E1 -18844.362,E2 -18844.362} C_VEL
LIN {X 0,Y 249.708,Z 440.384,A -85,B 0,C 180,E1 -18848.256,E2 -18848.256} C_VEL
LIN {X 0,Y 250.047,Z 438.579,A -85,B 0,C 180,E1 -18850.633,E2 -18850.633} C_VEL
LIN {X 0,Y 250.233,Z 436.828,A -85,B 0,C 180,E1 -18853.093,E2 -18853.093} C_VEL
LIN {X 0,Y 250.072,Z 434.259,A -85,B 0,C 180,E1 -18856.944,E2 -18856.944} C_VEL
LIN {X 0,Y 249.834,Z 432.566,A -85,B 0,C 180,E1 -18859.683,E2 -18859.683} C_VEL
LIN {X 0,Y 249.473,Z 430.279,A -85,B 0,C 180,E1 -18863.728,E2 -18863.728} C_VEL
LIN {X 0,Y 249.221,Z 428.21,A -85,B 0,C 180,E1 -18867.777,E2 -18867.777} C_VEL
LIN {X 0,Y 249.082,Z 426.96,A -85,B 0,C 180,E1 -18871.005,E2 -18871.005} C_VEL
LIN {X 0,Y 249.149,Z 426.955,A -85,B 0,C 180,E1 -18874.967,E2 -18874.967} C_VEL
LIN {X 0,Y 249.108,Z 426.958,A -85,B 0,C 180,E1 -18880.21,E2 -18880.21} C_VEL
LIN {X 0,Y 249.239,Z 426.938,A -85,B 0,C 180,E1 -18883.621,E2 -18883.621} C_VEL
LIN {X 0,Y 249.249,Z 426.939,A -85,B 0,C 180,E1 -18888.616,E2 -18888.616} C_VEL
LIN {X 0,Y 249.481,Z 426.908,A -85,B 0,C 180,E1 -18891.902,E2 -18891.902} C_VEL
LIN {X 0,Y 249.433,Z 426.915,A -85,B 0,C 180,E1 -18896.769,E2 -18896.769} C_VEL
LIN {X 0,Y 249.724,Z 426.869,A -85,B 0,C 180,E1 -18899.999,E2 -18899.999} C_VEL
LIN {X 0,Y 249.432,Z 426.901,A -85,B 0,C 180,E1 -18903.23,E2 -18903.23} C_VEL
LIN {X 0,Y 249.477,Z 426.91,A -85,B 0,C 180,E1 -18908.096,E2 -18908.096} C_VEL
LIN {X 0,Y 249.248,Z 426.935,A -85,B 0,C 180,E1 -18911.383,E2 -18911.383} C_VEL
LIN {X 0,Y 249.237,Z 426.94,A -85,B 0,C 180,E1 -18916.377,E2 -18916.377} C_VEL
LIN {X 0,Y 249.082,Z 426.956,A -85,B 0,C 180,E1 -18921.518,E2 -18921.518} C_VEL
LIN {X 0,Y 249.125,Z 426.947,A -85,B 0,C 180,E1 -18925.482,E2 -18925.482} C_VEL
LIN {X 0,Y 249.075,Z 426.957,A -85,B 0,C 180,E1 -18928.992,E2 -18928.992} C_VEL
LIN {X 0,Y 249.031,Z 426.964,A -85,B 0,C 180,E1 -18932.425,E2 -18932.425} C_VEL
LIN {X 0,Y 249.07,Z 426.96,A -85,B 0,C 180,E1 -18936.337,E2 -18936.337} C_VEL
LIN {X 0,Y 249.076,Z 426.957,A -85,B 0,C 180,E1 -18940.463,E2 -18940.463} C_VEL
LIN {X 0,Y 249.082,Z 426.956,A -85,B 0,C 180,E1 -18942.812,E2 -18942.812} C_VEL
LIN {X 0,Y 249.095,Z 426.957,A -85,B 0,C 180,E1 -18947.381,E2 -18947.381} C_VEL
LIN {X 0,Y 249.048,Z 426.964,A -85,B 0,C 180,E1 -18951.625,E2 -18951.625} C_VEL
LIN {X 0,Y 249.057,Z 426.963,A -85,B 0,C 180,E1 -18955.642,E2 -18955.642} C_VEL
LIN {X 0,Y 249.062,Z 426.979,A -85,B 0,C 180,E1 -18959.935,E2 -18959.935} C_VEL
LIN {X 0,Y 249.897,Z 429.526,A -85,B 0,C 180,E1 -18960.134,E2 -18960.134} C_VEL
LIN {X 0,Y 255.689,Z 440.685,A -85,B 0,C 180,E1 -18961.394,E2 -18961.394} C_VEL
LIN {X 0,Y 260.146,Z 451.297,A -85,B 0,C 180,E1 -18962.661,E2 -18962.661} C_VEL
LIN {X 0,Y 264.582,Z 461.116,A -85,B 0,C 180,E1 -18964.049,E2 -18964.049} C_VEL
LIN {X 0,Y 270.011,Z 470.326,A -85,B 0,C 180,E1 -18965.641,E2 -18965.641} C_VEL
LIN {X 0,Y 277.248,Z 480.245,A -85,B 0,C 180,E1 -18967.652,E2 -18967.652} C_VEL
LIN {X 0,Y 286.052,Z 490.394,A -85,B 0,C 180,E1 -18970.007,E2 -18970.007} C_VEL
LIN {X 0,Y 294.97,Z 499.582,A -85,B 0,C 180,E1 -18972.37,E2 -18972.37} C_VEL
LIN {X 0,Y 302.697,Z 506.997,A -85,B 0,C 180,E1 -18974.478,E2 -18974.478} C_VEL
LIN {X 0,Y 308.968,Z 512.872,A -85,B 0,C 180,E1 -18976.312,E2 -18976.312} C_VEL
LIN {X 0,Y 313.289,Z 516.756,A -85,B 0,C 180,E1 -18977.696,E2 -18977.696} C_VEL
LIN {X 0,Y 317.359,Z 520.439,A -85,B 0,C 180,E1 -18979.184,E2 -18979.184} C_VEL
LIN {X 0,Y 320.687,Z 523.059,A -85,B 0,C 180,E1 -18980.463,E2 -18980.463} C_VEL
LIN {X 0,Y 323.637,Z 525.634,A -85,B 0,C 180,E1 -18981.886,E2 -18981.886} C_VEL
LIN {X 0,Y 326.714,Z 528.358,A -85,B 0,C 180,E1 -18983.826,E2 -18983.826} C_VEL
LIN {X 0,Y 328.507,Z 529.651,A -85,B 0,C 180,E1 -18985.091,E2 -18985.091} C_VEL
LIN {X 0,Y 330.799,Z 530.874,A -85,B 0,C 180,E1 -18986.889,E2 -18986.889} C_VEL
LIN {X 0,Y 332.451,Z 531.453,A -85,B 0,C 180,E1 -18988.789,E2 -18988.789} C_VEL
LIN {X 0,Y 332.854,Z 531.524,A -85,B 0,C 180,E1 -18990,E2 -18990} C_VEL
LIN {X 0,Y 332.447,Z 531.444,A -85,B 0,C 180,E1 -18991.212,E2 -18991.212} C_VEL
LIN {X 0,Y 330.799,Z 530.864,A -85,B 0,C 180,E1 -18993.112,E2 -18993.112} C_VEL
LIN {X 0,Y 328.506,Z 529.664,A -85,B 0,C 180,E1 -18994.909,E2 -18994.909} C_VEL
LIN {X 0,Y 325.623,Z 527.495,A -85,B 0,C 180,E1 -18996.872,E2 -18996.872} C_VEL
LIN {X 0,Y 323.623,Z 525.651,A -85,B 0,C 180,E1 -18998.115,E2 -18998.115} C_VEL
LIN {X 0,Y 320.662,Z 523.087,A -85,B 0,C 180,E1 -18999.51,E2 -18999.51} C_VEL
LIN {X 0,Y 315.392,Z 518.677,A -85,B 0,C 180,E1 -19001.569,E2 -19001.569} C_VEL
LIN {X 0,Y 310.444,Z 514.191,A -85,B 0,C 180,E1 -19003.234,E2 -19003.234} C_VEL
LIN {X 0,Y 304.58,Z 508.621,A -85,B 0,C 180,E1 -19005.015,E2 -19005.015} C_VEL
LIN {X 0,Y 296.493,Z 501.038,A -85,B 0,C 180,E1 -19007.225,E2 -19007.225} C_VEL
LIN {X 0,Y 288.571,Z 493.085,A -85,B 0,C 180,E1 -19009.315,E2 -19009.315} C_VEL
LIN {X 0,Y 281.04,Z 484.756,A -85,B 0,C 180,E1 -19011.323,E2 -19011.323} C_VEL
LIN {X 0,Y 273.279,Z 475.107,A -85,B 0,C 180,E1 -19013.431,E2 -19013.431} C_VEL
LIN {X 0,Y 267.042,Z 465.508,A -85,B 0,C 180,E1 -19015.221,E2 -19015.221} C_VEL
LIN {X 0,Y 262.276,Z 456.364,A -85,B 0,C 180,E1 -19016.662,E2 -19016.662} C_VEL
LIN {X 0,Y 257.19,Z 444.073,A -85,B 0,C 180,E1 -19018.206,E2 -19018.206} C_VEL
LIN {X 0,Y 252.319,Z 433.842,A -85,B 0,C 180,E1 -19019.381,E2 -19019.381} C_VEL
LIN {X 0,Y 249.255,Z 427.987,A -85,B 0,C 180,E1 -19020.006,E2 -19020.006} C_VEL
LIN {X 0,Y 249.05,Z 426.963,A -85,B 0,C 180,E1 -19020.113,E2 -19020.113} C_VEL
LIN {X 0,Y 249.058,Z 426.963,A -85,B 0,C 180,E1 -19024.358,E2 -19024.358} C_VEL
LIN {X 0,Y 249.049,Z 426.964,A -85,B 0,C 180,E1 -19028.376,E2 -19028.376} C_VEL
LIN {X 0,Y 249.059,Z 426.961,A -85,B 0,C 180,E1 -19032.628,E2 -19032.628} C_VEL
LIN {X 0,Y 249.021,Z 426.963,A -85,B 0,C 180,E1 -19037.365,E2 -19037.365} C_VEL
LIN {X 0,Y 249.035,Z 426.963,A -85,B 0,C 180,E1 -19041.622,E2 -19041.622} C_VEL
LIN {X 0,Y 249.059,Z 426.961,A -85,B 0,C 180,E1 -19045.643,E2 -19045.643} C_VEL
LIN {X 0,Y 249.048,Z 426.961,A -85,B 0,C 180,E1 -19049.474,E2 -19049.474} C_VEL
LIN {X 0,Y 249.07,Z 426.958,A -85,B 0,C 180,E1 -19053.163,E2 -19053.163} C_VEL
LIN {X 0,Y 249.077,Z 426.957,A -85,B 0,C 180,E1 -19056.733,E2 -19056.733} C_VEL
LIN {X 0,Y 249.108,Z 426.952,A -85,B 0,C 180,E1 -19060.212,E2 -19060.212} C_VEL
LIN {X 0,Y 249.24,Z 426.939,A -85,B 0,C 180,E1 -19063.623,E2 -19063.623} C_VEL
LIN {X 0,Y 249.251,Z 426.935,A -85,B 0,C 180,E1 -19068.617,E2 -19068.617} C_VEL
LIN {X 0,Y 249.48,Z 426.91,A -85,B 0,C 180,E1 -19071.904,E2 -19071.904} C_VEL
LIN {X 0,Y 249.434,Z 426.9,A -85,B 0,C 180,E1 -19076.77,E2 -19076.77} C_VEL
LIN {X 0,Y 249.727,Z 426.868,A -85,B 0,C 180,E1 -19080.001,E2 -19080.001} C_VEL
LIN {X 0,Y 249.435,Z 426.914,A -85,B 0,C 180,E1 -19083.231,E2 -19083.231} C_VEL
LIN {X 0,Y 249.484,Z 426.907,A -85,B 0,C 180,E1 -19088.098,E2 -19088.098} C_VEL
LIN {X 0,Y 249.252,Z 426.939,A -85,B 0,C 180,E1 -19091.384,E2 -19091.384} C_VEL
LIN {X 0,Y 249.242,Z 426.937,A -85,B 0,C 180,E1 -19096.379,E2 -19096.379} C_VEL
LIN {X 0,Y 249.088,Z 426.959,A -85,B 0,C 180,E1 -19101.519,E2 -19101.519} C_VEL
LIN {X 0,Y 249.131,Z 426.953,A -85,B 0,C 180,E1 -19105.483,E2 -19105.483} C_VEL
LIN {X 0,Y 249.074,Z 426.962,A -85,B 0,C 180,E1 -19108.99,E2 -19108.99} C_VEL
LIN {X 0,Y 249.231,Z 428.295,A -85,B 0,C 180,E1 -19112.398,E2 -19112.398} C_VEL
LIN {X 0,Y 249.491,Z 430.279,A -85,B 0,C 180,E1 -19116.269,E2 -19116.269} C_VEL
LIN {X 0,Y 249.883,Z 432.749,A -85,B 0,C 180,E1 -19120.591,E2 -19120.591} C_VEL
LIN {X 0,Y 250.079,Z 434.264,A -85,B 0,C 180,E1 -19123.057,E2 -19123.057} C_VEL
LIN {X 0,Y 250.235,Z 436.85,A -85,B 0,C 180,E1 -19126.906,E2 -19126.906} C_VEL
LIN {X 0,Y 250.023,Z 438.901,A -85,B 0,C 180,E1 -19129.721,E2 -19129.721} C_VEL
LIN {X 0,Y 249.509,Z 441.288,A -85,B 0,C 180,E1 -19132.854,E2 -19132.854} C_VEL
LIN {X 0,Y 248.675,Z 442.059,A -85,B 0,C 180,E1 -19133.727,E2 -19133.727} C_VEL
LIN {X 0,Y 245.575,Z 443.439,A -85,B 0,C 180,E1 -19135.074,E2 -19135.074} C_VEL
LIN {X 0,Y 242.458,Z 444.792,A -85,B 0,C 180,E1 -19136.453,E2 -19136.453} C_VEL
LIN {X 0,Y 241.635,Z 445.561,A -85,B 0,C 180,E1 -19137.363,E2 -19137.363} C_VEL
LIN {X 0,Y 241.359,Z 447.181,A -85,B 0,C 180,E1 -19139.193,E2 -19139.193} C_VEL
LIN {X 0,Y 242.302,Z 450.446,A -85,B 0,C 180,E1 -19139.472,E2 -19139.472} C_VEL
LIN {X 0,Y 246.077,Z 463.268,A -85,B 0,C 180,E1 -19140.848,E2 -19140.848} C_VEL
LIN {X 0,Y 248.378,Z 474.107,A -85,B 0,C 180,E1 -19142.159,E2 -19142.159} C_VEL
LIN {X 0,Y 249.905,Z 484.419,A -85,B 0,C 180,E1 -19143.568,E2 -19143.568} C_VEL
LIN {X 0,Y 250.554,Z 493.401,A -85,B 0,C 180,E1 -19144.936,E2 -19144.936} C_VEL
LIN {X 0,Y 250.678,Z 502.167,A -85,B 0,C 180,E1 -19146.452,E2 -19146.452} C_VEL
LIN {X 0,Y 248.76,Z 510.697,A -85,B 0,C 180,E1 -19148.016,E2 -19148.016} C_VEL
LIN {X 0,Y 247.11,Z 517.918,A -85,B 0,C 180,E1 -19149.61,E2 -19149.61} C_VEL
LIN {X 0,Y 245.368,Z 525.502,A -85,B 0,C 180,E1 -19151.635,E2 -19151.635} C_VEL
LIN {X 0,Y 243.771,Z 531.82,A -85,B 0,C 180,E1 -19153.674,E2 -19153.674} C_VEL
LIN {X 0,Y 242.396,Z 537.083,A -85,B 0,C 180,E1 -19155.732,E2 -19155.732} C_VEL
LIN {X 0,Y 241.245,Z 542.218,A -85,B 0,C 180,E1 -19158.233,E2 -19158.233} C_VEL
LIN {X 0,Y 240.446,Z 546.212,A -85,B 0,C 180,E1 -19160.749,E2 -19160.749} C_VEL
LIN {X 0,Y 239.995,Z 549.168,A -85,B 0,C 180,E1 -19163.273,E2 -19163.273} C_VEL
LIN {X 0,Y 239.796,Z 551.624,A -85,B 0,C 180,E1 -19166.639,E2 -19166.639} C_VEL
LIN {X 0,Y 239.836,Z 552.217,A -85,B 0,C 180,E1 -19168.32,E2 -19168.32} C_VEL
LIN {X 0,Y 239.867,Z 552.373,A -85,B 0,C 180,E1 -19170,E2 -19170} C_VEL
LIN {X 0,Y 239.836,Z 552.217,A -85,B 0,C 180,E1 -19171.679,E2 -19171.679} C_VEL
LIN {X 0,Y 239.796,Z 551.624,A -85,B 0,C 180,E1 -19173.36,E2 -19173.36} C_VEL
LIN {X 0,Y 239.999,Z 549.169,A -85,B 0,C 180,E1 -19176.726,E2 -19176.726} C_VEL
LIN {X 0,Y 240.449,Z 546.213,A -85,B 0,C 180,E1 -19179.25,E2 -19179.25} C_VEL
LIN {X 0,Y 241.244,Z 542.22,A -85,B 0,C 180,E1 -19181.766,E2 -19181.766} C_VEL
LIN {X 0,Y 242.395,Z 537.085,A -85,B 0,C 180,E1 -19184.267,E2 -19184.267} C_VEL
LIN {X 0,Y 243.766,Z 531.822,A -85,B 0,C 180,E1 -19186.325,E2 -19186.325} C_VEL
LIN {X 0,Y 245.356,Z 525.504,A -85,B 0,C 180,E1 -19188.365,E2 -19188.365} C_VEL
LIN {X 0,Y 247.083,Z 517.92,A -85,B 0,C 180,E1 -19190.391,E2 -19190.391} C_VEL
LIN {X 0,Y 249.225,Z 508.781,A -85,B 0,C 180,E1 -19192.376,E2 -19192.376} C_VEL
LIN {X 0,Y 250.818,Z 501.033,A -85,B 0,C 180,E1 -19193.752,E2 -19193.752} C_VEL
LIN {X 0,Y 250.305,Z 489.044,A -85,B 0,C 180,E1 -19195.757,E2 -19195.757} C_VEL
LIN {X 0,Y 249.228,Z 479.672,A -85,B 0,C 180,E1 -19197.115,E2 -19197.115} C_VEL
LIN {X 0,Y 247.359,Z 468.992,A -85,B 0,C 180,E1 -19198.477,E2 -19198.477} C_VEL
LIN {X 0,Y 244.869,Z 458.985,A -85,B 0,C 180,E1 -19199.629,E2 -19199.629} C_VEL
LIN {X 0,Y 241.414,Z 447.764,A -85,B 0,C 180,E1 -19200.773,E2 -19200.773} C_VEL
LIN {X 0,Y 241.339,Z 447.016,A -85,B 0,C 180,E1 -19200.847,E2 -19200.847} C_VEL
LIN {X 0,Y 242.14,Z 443.259,A -85,B 0,C 180,E1 -19205.484,E2 -19205.484} C_VEL
LIN {X 0,Y 242.824,Z 440.193,A -85,B 0,C 180,E1 -19209.548,E2 -19209.548} C_VEL
LIN {X 0,Y 243.081,Z 438.671,A -85,B 0,C 180,E1 -19211.679,E2 -19211.679} C_VEL
LIN {X 0,Y 243.172,Z 437.151,A -85,B 0,C 180,E1 -19213.917,E2 -19213.917} C_VEL
LIN {X 0,Y 242.925,Z 434.38,A -85,B 0,C 180,E1 -19218.285,E2 -19218.285} C_VEL
LIN {X 0,Y 242.534,Z 431.977,A -85,B 0,C 180,E1 -19222.516,E2 -19222.516} C_VEL
LIN {X 0,Y 242.24,Z 429.528,A -85,B 0,C 180,E1 -19227.282,E2 -19227.282} C_VEL
LIN {X 0,Y 242.04,Z 428.035,A -85,B 0,C 180,E1 -19230.584,E2 -19230.584} C_VEL
LIN {X 0,Y 242.066,Z 427.837,A -85,B 0,C 180,E1 -19234.182,E2 -19234.182} C_VEL
LIN {X 0,Y 242.051,Z 427.839,A -85,B 0,C 180,E1 -19238.296,E2 -19238.296} C_VEL
LIN {X 0,Y 242.161,Z 427.82,A -85,B 0,C 180,E1 -19243.277,E2 -19243.277} C_VEL
LIN {X 0,Y 242.183,Z 427.819,A -85,B 0,C 180,E1 -19248.279,E2 -19248.279} C_VEL
LIN {X 0,Y 242.432,Z 427.785,A -85,B 0,C 180,E1 -19251.665,E2 -19251.665} C_VEL
LIN {X 0,Y 242.257,Z 427.808,A -85,B 0,C 180,E1 -19255.006,E2 -19255.006} C_VEL
LIN {X 0,Y 242.632,Z 427.759,A -85,B 0,C 180,E1 -19258.339,E2 -19258.339} C_VEL
LIN {X 0,Y 242.632,Z 427.74,A -85,B 0,C 180,E1 -19261.659,E2 -19261.659} C_VEL
LIN {X 0,Y 242.424,Z 427.787,A -85,B 0,C 180,E1 -19266.728,E2 -19266.728} C_VEL
LIN {X 0,Y 242.309,Z 427.798,A -85,B 0,C 180,E1 -19270.021,E2 -19270.021} C_VEL
LIN {X 0,Y 242.162,Z 427.814,A -85,B 0,C 180,E1 -19275.14,E2 -19275.14} C_VEL
LIN {X 0,Y 242.068,Z 427.829,A -85,B 0,C 180,E1 -19278.623,E2 -19278.623} C_VEL
LIN {X 0,Y 242.008,Z 427.841,A -85,B 0,C 180,E1 -19282.179,E2 -19282.179} C_VEL
LIN {X 0,Y 242.061,Z 427.828,A -85,B 0,C 180,E1 -19285.838,E2 -19285.838} C_VEL
LIN {X 0,Y 242.024,Z 427.837,A -85,B 0,C 180,E1 -19289.58,E2 -19289.58} C_VEL
LIN {X 0,Y 241.986,Z 427.842,A -85,B 0,C 180,E1 -19293.491,E2 -19293.491} C_VEL
LIN {X 0,Y 242.008,Z 427.841,A -85,B 0,C 180,E1 -19297.577,E2 -19297.577} C_VEL
LIN {X 0,Y 242.027,Z 427.838,A -85,B 0,C 180,E1 -19301.902,E2 -19301.902} C_VEL
LIN {X 0,Y 242.02,Z 427.837,A -85,B 0,C 180,E1 -19306.548,E2 -19306.548} C_VEL
LIN {X 0,Y 242.006,Z 427.84,A -85,B 0,C 180,E1 -19310.292,E2 -19310.292} C_VEL
LIN {X 0,Y 242.032,Z 427.836,A -85,B 0,C 180,E1 -19314.498,E2 -19314.498} C_VEL
LIN {X 0,Y 241.99,Z 427.843,A -85,B 0,C 180,E1 -19318.958,E2 -19318.958} C_VEL
LIN {X 0,Y 243.028,Z 430.729,A -85,B 0,C 180,E1 -19319.243,E2 -19319.243} C_VEL
LIN {X 0,Y 248.729,Z 441.59,A -85,B 0,C 180,E1 -19320.561,E2 -19320.561} C_VEL
LIN {X 0,Y 252.991,Z 451.523,A -85,B 0,C 180,E1 -19321.82,E2 -19321.82} C_VEL
LIN {X 0,Y 256.513,Z 460.277,A -85,B 0,C 180,E1 -19323.053,E2 -19323.053} C_VEL
LIN {X 0,Y 261.286,Z 469.65,A -85,B 0,C 180,E1 -19324.653,E2 -19324.653} C_VEL
LIN {X 0,Y 267.842,Z 479.655,A -85,B 0,C 180,E1 -19326.688,E2 -19326.688} C_VEL
LIN {X 0,Y 276.304,Z 490.012,A -85,B 0,C 180,E1 -19329.14,E2 -19329.14} C_VEL
LIN {X 0,Y 285.132,Z 499.25,A -85,B 0,C 180,E1 -19331.61,E2 -19331.61} C_VEL
LIN {X 0,Y 294.094,Z 507.745,A -85,B 0,C 180,E1 -19334.132,E2 -19334.132} C_VEL
LIN {X 0,Y 300.105,Z 513.084,A -85,B 0,C 180,E1 -19335.883,E2 -19335.883} C_VEL
LIN {X 0,Y 307.059,Z 519.269,A -85,B 0,C 180,E1 -19338.113,E2 -19338.113} C_VEL
LIN {X 0,Y 311.045,Z 522.799,A -85,B 0,C 180,E1 -19339.587,E2 -19339.587} C_VEL
LIN {X 0,Y 314.671,Z 525.718,A -85,B 0,C 180,E1 -19341.006,E2 -19341.006} C_VEL
LIN {X 0,Y 317.401,Z 528.078,A -85,B 0,C 180,E1 -19342.366,E2 -19342.366} C_VEL
LIN {X 0,Y 319.489,Z 529.912,A -85,B 0,C 180,E1 -19343.686,E2 -19343.686} C_VEL
LIN {X 0,Y 321.362,Z 531.403,A -85,B 0,C 180,E1 -19344.982,E2 -19344.982} C_VEL
LIN {X 0,Y 323.787,Z 532.796,A -85,B 0,C 180,E1 -19346.804,E2 -19346.804} C_VEL
LIN {X 0,Y 325.577,Z 533.452,A -85,B 0,C 180,E1 -19348.763,E2 -19348.763} C_VEL
LIN {X 0,Y 326.036,Z 533.526,A -85,B 0,C 180,E1 -19350,E2 -19350} C_VEL
LIN {X 0,Y 325.574,Z 533.444,A -85,B 0,C 180,E1 -19351.237,E2 -19351.237} C_VEL
LIN {X 0,Y 323.784,Z 532.793,A -85,B 0,C 180,E1 -19353.186,E2 -19353.186} C_VEL
LIN {X 0,Y 321.356,Z 531.395,A -85,B 0,C 180,E1 -19355.019,E2 -19355.019} C_VEL
LIN {X 0,Y 318.562,Z 529.156,A -85,B 0,C 180,E1 -19356.9,E2 -19356.9} C_VEL
LIN {X 0,Y 316.096,Z 526.986,A -85,B 0,C 180,E1 -19358.31,E2 -19358.31} C_VEL
LIN {X 0,Y 313.49,Z 524.783,A -85,B 0,C 180,E1 -19359.459,E2 -19359.459} C_VEL
LIN {X 0,Y 308.327,Z 520.385,A -85,B 0,C 180,E1 -19361.442,E2 -19361.442} C_VEL
LIN {X 0,Y 302.269,Z 515.015,A -85,B 0,C 180,E1 -19363.445,E2 -19363.445} C_VEL
LIN {X 0,Y 295.42,Z 508.903,A -85,B 0,C 180,E1 -19365.492,E2 -19365.492} C_VEL
LIN {X 0,Y 286.401,Z 500.524,A -85,B 0,C 180,E1 -19368.035,E2 -19368.035} C_VEL
LIN {X 0,Y 277.582,Z 491.457,A -85,B 0,C 180,E1 -19370.484,E2 -19370.484} C_VEL
LIN {X 0,Y 269.048,Z 481.192,A -85,B 0,C 180,E1 -19372.962,E2 -19372.962} C_VEL
LIN {X 0,Y 262.513,Z 471.678,A -85,B 0,C 180,E1 -19374.956,E2 -19374.956} C_VEL
LIN {X 0,Y 258.03,Z 463.569,A -85,B 0,C 180,E1 -19376.416,E2 -19376.416} C_VEL
LIN {X 0,Y 254.163,Z 454.559,A -85,B 0,C 180,E1 -19377.769,E2 -19377.769} C_VEL
LIN {X 0,Y 249.739,Z 443.776,A -85,B 0,C 180,E1 -19379.162,E2 -19379.162} C_VEL
LIN {X 0,Y 244.539,Z 433.476,A -85,B 0,C 180,E1 -19380.438,E2 -19380.438} C_VEL
LIN {X 0,Y 242.139,Z 428.677,A -85,B 0,C 180,E1 -19380.968,E2 -19380.968} C_VEL
LIN {X 0,Y 241.98,Z 427.844,A -85,B 0,C 180,E1 -19381.067,E2 -19381.067} C_VEL
LIN {X 0,Y 242.026,Z 427.837,A -85,B 0,C 180,E1 -19385.605,E2 -19385.605} C_VEL
LIN {X 0,Y 242.005,Z 427.84,A -85,B 0,C 180,E1 -19389.709,E2 -19389.709} C_VEL
LIN {X 0,Y 241.974,Z 427.845,A -85,B 0,C 180,E1 -19394.192,E2 -19394.192} C_VEL
LIN {X 0,Y 241.948,Z 427.845,A -85,B 0,C 180,E1 -19399.046,E2 -19399.046} C_VEL
LIN {X 0,Y 241.999,Z 427.842,A -85,B 0,C 180,E1 -19402.421,E2 -19402.421} C_VEL
LIN {X 0,Y 241.989,Z 427.842,A -85,B 0,C 180,E1 -19406.51,E2 -19406.51} C_VEL
LIN {X 0,Y 242.033,Z 427.835,A -85,B 0,C 180,E1 -19410.588,E2 -19410.588} C_VEL
LIN {X 0,Y 242.065,Z 427.828,A -85,B 0,C 180,E1 -19414.184,E2 -19414.184} C_VEL
LIN {X 0,Y 242.051,Z 427.832,A -85,B 0,C 180,E1 -19418.298,E2 -19418.298} C_VEL
LIN {X 0,Y 242.161,Z 427.82,A -85,B 0,C 180,E1 -19423.279,E2 -19423.279} C_VEL
LIN {X 0,Y 242.184,Z 427.816,A -85,B 0,C 180,E1 -19428.281,E2 -19428.281} C_VEL
LIN {X 0,Y 242.426,Z 427.786,A -85,B 0,C 180,E1 -19431.666,E2 -19431.666} C_VEL
LIN {X 0,Y 242.259,Z 427.804,A -85,B 0,C 180,E1 -19435.008,E2 -19435.008} C_VEL
LIN {X 0,Y 242.635,Z 427.74,A -85,B 0,C 180,E1 -19438.341,E2 -19438.341} C_VEL
LIN {X 0,Y 242.635,Z 427.759,A -85,B 0,C 180,E1 -19441.661,E2 -19441.661} C_VEL
LIN {X 0,Y 242.433,Z 427.784,A -85,B 0,C 180,E1 -19446.66,E2 -19446.66} C_VEL
LIN {X 0,Y 242.345,Z 427.797,A -85,B 0,C 180,E1 -19450.021,E2 -19450.021} C_VEL
LIN {X 0,Y 242.166,Z 427.821,A -85,B 0,C 180,E1 -19455.142,E2 -19455.142} C_VEL
LIN {X 0,Y 242.073,Z 427.831,A -85,B 0,C 180,E1 -19458.625,E2 -19458.625} C_VEL
LIN {X 0,Y 242.013,Z 427.838,A -85,B 0,C 180,E1 -19462.181,E2 -19462.181} C_VEL
LIN {X 0,Y 242.067,Z 427.831,A -85,B 0,C 180,E1 -19465.839,E2 -19465.839} C_VEL
LIN {X 0,Y 242.036,Z 428.11,A -85,B 0,C 180,E1 -19469.58,E2 -19469.58} C_VEL
LIN {X 0,Y 242.256,Z 429.911,A -85,B 0,C 180,E1 -19473.451,E2 -19473.451} C_VEL
LIN {X 0,Y 242.55,Z 431.977,A -85,B 0,C 180,E1 -19477.481,E2 -19477.481} C_VEL
LIN {X 0,Y 242.929,Z 434.396,A -85,B 0,C 180,E1 -19481.714,E2 -19481.714} C_VEL
LIN {X 0,Y 243.174,Z 437.157,A -85,B 0,C 180,E1 -19486.082,E2 -19486.082} C_VEL
LIN {X 0,Y 243.059,Z 439.002,A -85,B 0,C 180,E1 -19488.747,E2 -19488.747} C_VEL
LIN {X 0,Y 242.449,Z 441.96,A -85,B 0,C 180,E1 -19492.742,E2 -19492.742} C_VEL
LIN {X 0,Y 241.797,Z 444.869,A -85,B 0,C 180,E1 -19496.479,E2 -19496.479} C_VEL
LIN {X 0,Y 241.635,Z 445.561,A -85,B 0,C 180,E1 -19497.363,E2 -19497.363} C_VEL
LIN {X 0,Y 241.513,Z 447.062,A -85,B 0,C 180,E1 -19498.166,E2 -19498.166} C_VEL
LIN {X 0,Y 241.405,Z 449.665,A -85,B 0,C 180,E1 -19498.814,E2 -19498.814} C_VEL
LIN {X 0,Y 241.231,Z 454.732,A -85,B 0,C 180,E1 -19499.533,E2 -19499.533} C_VEL
LIN {X 0,Y 241.177,Z 470.954,A -85,B 0,C 180,E1 -19500.921,E2 -19500.921} C_VEL
LIN {X 0,Y 241.411,Z 472.851,A -85,B 0,C 180,E1 -19501.163,E2 -19501.163} C_VEL
LIN {X 0,Y 243.017,Z 483.357,A -85,B 0,C 180,E1 -19502.64,E2 -19502.64} C_VEL
LIN {X 0,Y 243.834,Z 493.147,A -85,B 0,C 180,E1 -19504.19,E2 -19504.19} C_VEL
LIN {X 0,Y 243.988,Z 501.949,A -85,B 0,C 180,E1 -19505.766,E2 -19505.766} C_VEL
LIN {X 0,Y 242.663,Z 508.566,A -85,B 0,C 180,E1 -19506.984,E2 -19506.984} C_VEL
LIN {X 0,Y 240.421,Z 517.705,A -85,B 0,C 180,E1 -19509.017,E2 -19509.017} C_VEL
LIN {X 0,Y 239.129,Z 523.583,A -85,B 0,C 180,E1 -19510.585,E2 -19510.585} C_VEL
LIN {X 0,Y 237.226,Z 530.452,A -85,B 0,C 180,E1 -19512.767,E2 -19512.767} C_VEL
LIN {X 0,Y 236.037,Z 534.955,A -85,B 0,C 180,E1 -19514.456,E2 -19514.456} C_VEL
LIN {X 0,Y 234.617,Z 540.45,A -85,B 0,C 180,E1 -19517.017,E2 -19517.017} C_VEL
LIN {X 0,Y 233.68,Z 544.782,A -85,B 0,C 180,E1 -19519.604,E2 -19519.604} C_VEL
LIN {X 0,Y 233.214,Z 547.152,A -85,B 0,C 180,E1 -19521.334,E2 -19521.334} C_VEL
LIN {X 0,Y 232.922,Z 548.956,A -85,B 0,C 180,E1 -19523.068,E2 -19523.068} C_VEL
LIN {X 0,Y 232.705,Z 551.412,A -85,B 0,C 180,E1 -19526.537,E2 -19526.537} C_VEL
LIN {X 0,Y 232.749,Z 552.006,A -85,B 0,C 180,E1 -19528.269,E2 -19528.269} C_VEL
LIN {X 0,Y 232.779,Z 552.162,A -85,B 0,C 180,E1 -19530,E2 -19530} C_VEL
LIN {X 0,Y 232.749,Z 552.006,A -85,B 0,C 180,E1 -19531.73,E2 -19531.73} C_VEL
LIN {X 0,Y 232.757,Z 550.595,A -85,B 0,C 180,E1 -19534.839,E2 -19534.839} C_VEL
LIN {X 0,Y 232.925,Z 548.957,A -85,B 0,C 180,E1 -19536.932,E2 -19536.932} C_VEL
LIN {X 0,Y 233.426,Z 546.002,A -85,B 0,C 180,E1 -19539.531,E2 -19539.531} C_VEL
LIN {X 0,Y 234.276,Z 542.008,A -85,B 0,C 180,E1 -19542.121,E2 -19542.121} C_VEL
LIN {X 0,Y 235.492,Z 536.873,A -85,B 0,C 180,E1 -19544.694,E2 -19544.694} C_VEL
LIN {X 0,Y 236.935,Z 531.61,A -85,B 0,C 180,E1 -19546.81,E2 -19546.81} C_VEL
LIN {X 0,Y 238.623,Z 525.292,A -85,B 0,C 180,E1 -19548.903,E2 -19548.903} C_VEL
LIN {X 0,Y 240.038,Z 519.336,A -85,B 0,C 180,E1 -19550.569,E2 -19550.569} C_VEL
LIN {X 0,Y 241.692,Z 512.407,A -85,B 0,C 180,E1 -19552.21,E2 -19552.21} C_VEL
LIN {X 0,Y 243.646,Z 504.228,A -85,B 0,C 180,E1 -19553.817,E2 -19553.817} C_VEL
LIN {X 0,Y 244.078,Z 499.662,A -85,B 0,C 180,E1 -19554.677,E2 -19554.677} C_VEL
LIN {X 0,Y 243.535,Z 488.733,A -85,B 0,C 180,E1 -19556.54,E2 -19556.54} C_VEL
LIN {X 0,Y 242.243,Z 477.785,A -85,B 0,C 180,E1 -19558.157,E2 -19558.157} C_VEL
LIN {X 0,Y 240.501,Z 468.384,A -85,B 0,C 180,E1 -19559.401,E2 -19559.401} C_VEL
LIN {X 0,Y 237.702,Z 457.624,A -85,B 0,C 180,E1 -19560.695,E2 -19560.695} C_VEL
LIN {X 0,Y 234.554,Z 447.858,A -85,B 0,C 180,E1 -19561.76,E2 -19561.76} C_VEL
LIN {X 0,Y 234.422,Z 446.812,A -85,B 0,C 180,E1 -19561.858,E2 -19561.858} C_VEL
LIN {X 0,Y 235.156,Z 443.432,A -85,B 0,C 180,E1 -19566.201,E2 -19566.201} C_VEL
LIN {X 0,Y 235.707,Z 441.279,A -85,B 0,C 180,E1 -19569.172,E2 -19569.172} C_VEL
LIN {X 0,Y 236.04,Z 439.371,A -85,B 0,C 180,E1 -19571.894,E2 -19571.894} C_VEL
LIN {X 0,Y 236.038,Z 436.948,A -85,B 0,C 180,E1 -19575.609,E2 -19575.609} C_VEL
LIN {X 0,Y 235.83,Z 434.905,A -85,B 0,C 180,E1 -19579.032,E2 -19579.032} C_VEL
LIN {X 0,Y 235.416,Z 432.376,A -85,B 0,C 180,E1 -19583.71,E2 -19583.71} C_VEL
LIN {X 0,Y 235.205,Z 430.539,A -85,B 0,C 180,E1 -19587.462,E2 -19587.462} C_VEL
LIN {X 0,Y 234.952,Z 428.821,A -85,B 0,C 180,E1 -19591.405,E2 -19591.405} C_VEL
LIN {X 0,Y 234.985,Z 428.72,A -85,B 0,C 180,E1 -19595.246,E2 -19595.246} C_VEL
LIN {X 0,Y 235.009,Z 428.716,A -85,B 0,C 180,E1 -19598.969,E2 -19598.969} C_VEL
LIN {X 0,Y 235.094,Z 428.702,A -85,B 0,C 180,E1 -19603.058,E2 -19603.058} C_VEL
LIN {X 0,Y 235.115,Z 428.698,A -85,B 0,C 180,E1 -19607.921,E2 -19607.921} C_VEL
LIN {X 0,Y 235.387,Z 428.663,A -85,B 0,C 180,E1 -19611.414,E2 -19611.414} C_VEL
LIN {X 0,Y 235.402,Z 428.662,A -85,B 0,C 180,E1 -19613.14,E2 -19613.14} C_VEL
LIN {X 0,Y 235.592,Z 428.637,A -85,B 0,C 180,E1 -19618.29,E2 -19618.29} C_VEL
LIN {X 0,Y 235.592,Z 428.616,A -85,B 0,C 180,E1 -19621.709,E2 -19621.709} C_VEL
LIN {X 0,Y 235.4,Z 428.662,A -85,B 0,C 180,E1 -19626.858,E2 -19626.858} C_VEL
LIN {X 0,Y 235.233,Z 428.68,A -85,B 0,C 180,E1 -19630.326,E2 -19630.326} C_VEL
LIN {X 0,Y 235.109,Z 428.693,A -85,B 0,C 180,E1 -19635.606,E2 -19635.606} C_VEL
LIN {X 0,Y 235.003,Z 428.708,A -85,B 0,C 180,E1 -19639.205,E2 -19639.205} C_VEL
LIN {X 0,Y 234.956,Z 428.716,A -85,B 0,C 180,E1 -19642.882,E2 -19642.882} C_VEL
LIN {X 0,Y 234.964,Z 428.716,A -85,B 0,C 180,E1 -19646.657,E2 -19646.657} C_VEL
LIN {X 0,Y 234.926,Z 428.72,A -85,B 0,C 180,E1 -19650.567,E2 -19650.567} C_VEL
LIN {X 0,Y 234.955,Z 428.717,A -85,B 0,C 180,E1 -19654.633,E2 -19654.633} C_VEL
LIN {X 0,Y 234.961,Z 428.716,A -85,B 0,C 180,E1 -19658.952,E2 -19658.952} C_VEL
LIN {X 0,Y 234.988,Z 428.714,A -85,B 0,C 180,E1 -19663.461,E2 -19663.461} C_VEL
LIN {X 0,Y 234.992,Z 428.712,A -85,B 0,C 180,E1 -19666.54,E2 -19666.54} C_VEL
LIN {X 0,Y 234.95,Z 428.719,A -85,B 0,C 180,E1 -19671.086,E2 -19671.086} C_VEL
LIN {X 0,Y 234.956,Z 428.719,A -85,B 0,C 180,E1 -19675.367,E2 -19675.367} C_VEL
LIN {X 0,Y 234.952,Z 428.8,A -85,B 0,C 180,E1 -19677.97,E2 -19677.97} C_VEL
LIN {X 0,Y 235.878,Z 431.492,A -85,B 0,C 180,E1 -19678.228,E2 -19678.228} C_VEL
LIN {X 0,Y 238.652,Z 436.354,A -85,B 0,C 180,E1 -19678.863,E2 -19678.863} C_VEL
LIN {X 0,Y 244.422,Z 448.238,A -85,B 0,C 180,E1 -19680.439,E2 -19680.439} C_VEL
LIN {X 0,Y 249.275,Z 460.741,A -85,B 0,C 180,E1 -19682.228,E2 -19682.228} C_VEL
LIN {X 0,Y 253.441,Z 469.934,A -85,B 0,C 180,E1 -19683.812,E2 -19683.812} C_VEL
LIN {X 0,Y 258.369,Z 478.417,A -85,B 0,C 180,E1 -19685.547,E2 -19685.547} C_VEL
LIN {X 0,Y 265.557,Z 488.186,A -85,B 0,C 180,E1 -19687.86,E2 -19687.86} C_VEL
LIN {X 0,Y 275.323,Z 499.018,A -85,B 0,C 180,E1 -19690.815,E2 -19690.815} C_VEL
LIN {X 0,Y 284.172,Z 507.418,A -85,B 0,C 180,E1 -19693.4,E2 -19693.4} C_VEL
LIN {X 0,Y 292.326,Z 514.416,A -85,B 0,C 180,E1 -19695.815,E2 -19695.815} C_VEL
LIN {X 0,Y 298.383,Z 519.534,A -85,B 0,C 180,E1 -19697.762,E2 -19697.762} C_VEL
LIN {X 0,Y 304.696,Z 524.784,A -85,B 0,C 180,E1 -19700.039,E2 -19700.039} C_VEL
LIN {X 0,Y 308.319,Z 527.61,A -85,B 0,C 180,E1 -19701.48,E2 -19701.48} C_VEL
LIN {X 0,Y 311.451,Z 530.337,A -85,B 0,C 180,E1 -19703.149,E2 -19703.149} C_VEL
LIN {X 0,Y 314.022,Z 532.524,A -85,B 0,C 180,E1 -19704.864,E2 -19704.864} C_VEL
LIN {X 0,Y 316.734,Z 534.171,A -85,B 0,C 180,E1 -19706.848,E2 -19706.848} C_VEL
LIN {X 0,Y 318.527,Z 534.839,A -85,B 0,C 180,E1 -19708.736,E2 -19708.736} C_VEL
LIN {X 0,Y 319.063,Z 534.948,A -85,B 0,C 180,E1 -19710,E2 -19710} C_VEL
LIN {X 0,Y 318.525,Z 534.835,A -85,B 0,C 180,E1 -19711.265,E2 -19711.265} C_VEL
LIN {X 0,Y 316.732,Z 534.166,A -85,B 0,C 180,E1 -19713.146,E2 -19713.146} C_VEL
LIN {X 0,Y 314.009,Z 532.511,A -85,B 0,C 180,E1 -19715.137,E2 -19715.137} C_VEL
LIN {X 0,Y 311.441,Z 530.358,A -85,B 0,C 180,E1 -19716.835,E2 -19716.835} C_VEL
LIN {X 0,Y 308.248,Z 527.612,A -85,B 0,C 180,E1 -19718.523,E2 -19718.523} C_VEL
LIN {X 0,Y 302.775,Z 523.142,A -85,B 0,C 180,E1 -19720.702,E2 -19720.702} C_VEL
LIN {X 0,Y 296.687,Z 518.071,A -85,B 0,C 180,E1 -19722.807,E2 -19722.807} C_VEL
LIN {X 0,Y 290.627,Z 512.976,A -85,B 0,C 180,E1 -19724.699,E2 -19724.699} C_VEL
LIN {X 0,Y 281.309,Z 504.751,A -85,B 0,C 180,E1 -19727.446,E2 -19727.446} C_VEL
LIN {X 0,Y 272.129,Z 495.698,A -85,B 0,C 180,E1 -19730.136,E2 -19730.136} C_VEL
LIN {X 0,Y 264.511,Z 486.849,A -85,B 0,C 180,E1 -19732.469,E2 -19732.469} C_VEL
LIN {X 0,Y 258.361,Z 478.372,A -85,B 0,C 180,E1 -19734.465,E2 -19734.465} C_VEL
LIN {X 0,Y 252.837,Z 468.774,A -85,B 0,C 180,E1 -19736.407,E2 -19736.407} C_VEL
LIN {X 0,Y 248.482,Z 458.697,A -85,B 0,C 180,E1 -19738.087,E2 -19738.087} C_VEL
LIN {X 0,Y 243.574,Z 446.348,A -85,B 0,C 180,E1 -19739.812,E2 -19739.812} C_VEL
LIN {X 0,Y 237.905,Z 435.02,A -85,B 0,C 180,E1 -19741.322,E2 -19741.322} C_VEL
LIN {X 0,Y 236.036,Z 431.741,A -85,B 0,C 180,E1 -19741.745,E2 -19741.745} C_VEL
LIN {X 0,Y 234.942,Z 428.72,A -85,B 0,C 180,E1 -19742.08,E2 -19742.08} C_VEL
LIN {X 0,Y 234.954,Z 428.719,A -85,B 0,C 180,E1 -19746.137,E2 -19746.137} C_VEL
LIN {X 0,Y 234.964,Z 428.717,A -85,B 0,C 180,E1 -19748.952,E2 -19748.952} C_VEL
LIN {X 0,Y 234.962,Z 428.716,A -85,B 0,C 180,E1 -19753.468,E2 -19753.468} C_VEL
LIN {X 0,Y 234.919,Z 428.723,A -85,B 0,C 180,E1 -19758.41,E2 -19758.41} C_VEL
LIN {X 0,Y 234.952,Z 428.717,A -85,B 0,C 180,E1 -19761.087,E2 -19761.087} C_VEL
LIN {X 0,Y 234.958,Z 428.717,A -85,B 0,C 180,E1 -19765.368,E2 -19765.368} C_VEL
LIN {X 0,Y 234.966,Z 428.718,A -85,B 0,C 180,E1 -19770.158,E2 -19770.158} C_VEL
LIN {X 0,Y 234.992,Z 428.712,A -85,B 0,C 180,E1 -19773.795,E2 -19773.795} C_VEL
LIN {X 0,Y 235.009,Z 428.708,A -85,B 0,C 180,E1 -19778.971,E2 -19778.971} C_VEL
LIN {X 0,Y 235.094,Z 428.699,A -85,B 0,C 180,E1 -19783.06,E2 -19783.06} C_VEL
LIN {X 0,Y 235.145,Z 428.695,A -85,B 0,C 180,E1 -19787.925,E2 -19787.925} C_VEL
LIN {X 0,Y 235.375,Z 428.662,A -85,B 0,C 180,E1 -19791.415,E2 -19791.415} C_VEL
LIN {X 0,Y 235.403,Z 428.662,A -85,B 0,C 180,E1 -19793.142,E2 -19793.142} C_VEL
LIN {X 0,Y 235.594,Z 428.615,A -85,B 0,C 180,E1 -19798.292,E2 -19798.292} C_VEL
LIN {X 0,Y 235.595,Z 428.636,A -85,B 0,C 180,E1 -19801.71,E2 -19801.71} C_VEL
LIN {X 0,Y 235.405,Z 428.66,A -85,B 0,C 180,E1 -19806.86,E2 -19806.86} C_VEL
LIN {X 0,Y 235.253,Z 428.68,A -85,B 0,C 180,E1 -19810.327,E2 -19810.327} C_VEL
LIN {X 0,Y 235.114,Z 428.699,A -85,B 0,C 180,E1 -19815.607,E2 -19815.607} C_VEL
LIN {X 0,Y 235.009,Z 428.713,A -85,B 0,C 180,E1 -19819.206,E2 -19819.206} C_VEL
LIN {X 0,Y 234.962,Z 428.718,A -85,B 0,C 180,E1 -19822.884,E2 -19822.884} C_VEL
LIN {X 0,Y 234.968,Z 428.716,A -85,B 0,C 180,E1 -19826.658,E2 -19826.658} C_VEL
LIN {X 0,Y 234.949,Z 428.823,A -85,B 0,C 180,E1 -19828.595,E2 -19828.595} C_VEL
LIN {X 0,Y 235.24,Z 430.866,A -85,B 0,C 180,E1 -19833.226,E2 -19833.226} C_VEL
LIN {X 0,Y 235.448,Z 432.575,A -85,B 0,C 180,E1 -19836.656,E2 -19836.656} C_VEL
LIN {X 0,Y 235.835,Z 434.921,A -85,B 0,C 180,E1 -19840.967,E2 -19840.967} C_VEL
LIN {X 0,Y 236.043,Z 436.97,A -85,B 0,C 180,E1 -19844.391,E2 -19844.391} C_VEL
LIN {X 0,Y 236.054,Z 439.375,A -85,B 0,C 180,E1 -19848.102,E2 -19848.102} C_VEL
LIN {X 0,Y 235.667,Z 441.592,A -85,B 0,C 180,E1 -19851.226,E2 -19851.226} C_VEL
LIN {X 0,Y 234.911,Z 444.657,A -85,B 0,C 180,E1 -19855.359,E2 -19855.359} C_VEL
LIN {X 0,Y 234.435,Z 446.803,A -85,B 0,C 180,E1 -19858.143,E2 -19858.143} C_VEL
LIN {X 0,Y 235.424,Z 450.333,A -85,B 0,C 180,E1 -19858.486,E2 -19858.486} C_VEL
LIN {X 0,Y 239.516,Z 464.204,A -85,B 0,C 180,E1 -19860.078,E2 -19860.078} C_VEL
LIN {X 0,Y 241.411,Z 472.851,A -85,B 0,C 180,E1 -19861.163,E2 -19861.163} C_VEL
LIN {X 0,Y 241.708,Z 476.455,A -85,B 0,C 180,E1 -19861.613,E2 -19861.613} C_VEL
LIN {X 0,Y 241.204,Z 481.927,A -85,B 0,C 180,E1 -19862.221,E2 -19862.221} C_VEL
LIN {X 0,Y 237.884,Z 495.585,A -85,B 0,C 180,E1 -19863.92,E2 -19863.92} C_VEL
LIN {X 0,Y 237.293,Z 500.377,A -85,B 0,C 180,E1 -19864.759,E2 -19864.759} C_VEL
LIN {X 0,Y 236.922,Z 505.148,A -85,B 0,C 180,E1 -19865.696,E2 -19865.696} C_VEL
LIN {X 0,Y 234.201,Z 515.865,A -85,B 0,C 180,E1 -19867.969,E2 -19867.969} C_VEL
LIN {X 0,Y 232.329,Z 523.671,A -85,B 0,C 180,E1 -19870.093,E2 -19870.093} C_VEL
LIN {X 0,Y 230.405,Z 530.239,A -85,B 0,C 180,E1 -19872.24,E2 -19872.24} C_VEL
LIN {X 0,Y 229.174,Z 534.743,A -85,B 0,C 180,E1 -19873.978,E2 -19873.978} C_VEL
LIN {X 0,Y 227.672,Z 540.238,A -85,B 0,C 180,E1 -19876.613,E2 -19876.613} C_VEL
LIN {X 0,Y 226.661,Z 544.569,A -85,B 0,C 180,E1 -19879.278,E2 -19879.278} C_VEL
LIN {X 0,Y 226.171,Z 546.94,A -85,B 0,C 180,E1 -19881.062,E2 -19881.062} C_VEL
LIN {X 0,Y 225.847,Z 548.744,A -85,B 0,C 180,E1 -19882.849,E2 -19882.849} C_VEL
LIN {X 0,Y 225.617,Z 551.201,A -85,B 0,C 180,E1 -19886.428,E2 -19886.428} C_VEL
LIN {X 0,Y 225.664,Z 551.795,A -85,B 0,C 180,E1 -19888.215,E2 -19888.215} C_VEL
LIN {X 0,Y 225.693,Z 551.952,A -85,B 0,C 180,E1 -19890,E2 -19890} C_VEL
LIN {X 0,Y 225.664,Z 551.795,A -85,B 0,C 180,E1 -19891.784,E2 -19891.784} C_VEL
LIN {X 0,Y 225.668,Z 550.556,A -85,B 0,C 180,E1 -19894.731,E2 -19894.731} C_VEL
LIN {X 0,Y 225.85,Z 548.745,A -85,B 0,C 180,E1 -19897.15,E2 -19897.15} C_VEL
LIN {X 0,Y 226.392,Z 545.789,A -85,B 0,C 180,E1 -19899.83,E2 -19899.83} C_VEL
LIN {X 0,Y 227.301,Z 541.795,A -85,B 0,C 180,E1 -19902.499,E2 -19902.499} C_VEL
LIN {X 0,Y 228.607,Z 536.661,A -85,B 0,C 180,E1 -19905.147,E2 -19905.147} C_VEL
LIN {X 0,Y 230.118,Z 531.398,A -85,B 0,C 180,E1 -19907.323,E2 -19907.323} C_VEL
LIN {X 0,Y 231.898,Z 525.081,A -85,B 0,C 180,E1 -19909.473,E2 -19909.473} C_VEL
LIN {X 0,Y 233.369,Z 519.124,A -85,B 0,C 180,E1 -19911.185,E2 -19911.185} C_VEL
LIN {X 0,Y 235.123,Z 512.195,A -85,B 0,C 180,E1 -19912.865,E2 -19912.865} C_VEL
LIN {X 0,Y 237.159,Z 504.017,A -85,B 0,C 180,E1 -19914.511,E2 -19914.511} C_VEL
LIN {X 0,Y 237.28,Z 496.808,A -85,B 0,C 180,E1 -19915.904,E2 -19915.904} C_VEL
LIN {X 0,Y 236.796,Z 487.633,A -85,B 0,C 180,E1 -19917.485,E2 -19917.485} C_VEL
LIN {X 0,Y 235.532,Z 477.558,A -85,B 0,C 180,E1 -19919.034,E2 -19919.034} C_VEL
LIN {X 0,Y 233.739,Z 468.269,A -85,B 0,C 180,E1 -19920.328,E2 -19920.328} C_VEL
LIN {X 0,Y 230.886,Z 457.489,A -85,B 0,C 180,E1 -19921.697,E2 -19921.697} C_VEL
LIN {X 0,Y 228.189,Z 449.377,A -85,B 0,C 180,E1 -19922.669,E2 -19922.669} C_VEL
LIN {X 0,Y 227.537,Z 446.623,A -85,B 0,C 180,E1 -19922.918,E2 -19922.918} C_VEL
LIN {X 0,Y 228.398,Z 442.887,A -85,B 0,C 180,E1 -19927.981,E2 -19927.981} C_VEL
LIN {X 0,Y 228.759,Z 441.367,A -85,B 0,C 180,E1 -19930.177,E2 -19930.177} C_VEL
LIN {X 0,Y 229.021,Z 439.767,A -85,B 0,C 180,E1 -19932.565,E2 -19932.565} C_VEL
LIN {X 0,Y 229.005,Z 438.154,A -85,B 0,C 180,E1 -19935.1,E2 -19935.1} C_VEL
LIN {X 0,Y 228.88,Z 436.741,A -85,B 0,C 180,E1 -19937.503,E2 -19937.503} C_VEL
LIN {X 0,Y 228.656,Z 435.234,A -85,B 0,C 180,E1 -19940.209,E2 -19940.209} C_VEL
LIN {X 0,Y 228.357,Z 433.161,A -85,B 0,C 180,E1 -19944.214,E2 -19944.214} C_VEL
LIN {X 0,Y 228.116,Z 431.197,A -85,B 0,C 180,E1 -19948.415,E2 -19948.415} C_VEL
LIN {X 0,Y 227.885,Z 429.602,A -85,B 0,C 180,E1 -19952.444,E2 -19952.444} C_VEL
LIN {X 0,Y 227.912,Z 429.601,A -85,B 0,C 180,E1 -19956.366,E2 -19956.366} C_VEL
LIN {X 0,Y 227.94,Z 429.595,A -85,B 0,C 180,E1 -19960.173,E2 -19960.173} C_VEL
LIN {X 0,Y 228.055,Z 429.577,A -85,B 0,C 180,E1 -19963.897,E2 -19963.897} C_VEL
LIN {X 0,Y 228.072,Z 429.575,A -85,B 0,C 180,E1 -19967.542,E2 -19967.542} C_VEL
LIN {X 0,Y 228.322,Z 429.544,A -85,B 0,C 180,E1 -19971.146,E2 -19971.146} C_VEL
LIN {X 0,Y 228.355,Z 429.541,A -85,B 0,C 180,E1 -19972.928,E2 -19972.928} C_VEL
LIN {X 0,Y 228.551,Z 429.514,A -85,B 0,C 180,E1 -19978.237,E2 -19978.237} C_VEL
LIN {X 0,Y 228.55,Z 429.491,A -85,B 0,C 180,E1 -19981.761,E2 -19981.761} C_VEL
LIN {X 0,Y 228.351,Z 429.54,A -85,B 0,C 180,E1 -19987.071,E2 -19987.071} C_VEL
LIN {X 0,Y 228.159,Z 429.562,A -85,B 0,C 180,E1 -19990.65,E2 -19990.65} C_VEL
LIN {X 0,Y 228.06,Z 429.572,A -85,B 0,C 180,E1 -19994.271,E2 -19994.271} C_VEL
LIN {X 0,Y 227.998,Z 429.586,A -85,B 0,C 180,E1 -19997.953,E2 -19997.953} C_VEL
LIN {X 0,Y 227.925,Z 429.594,A -85,B 0,C 180,E1 -20002.329,E2 -20002.329} C_VEL
LIN {X 0,Y 227.938,Z 429.591,A -85,B 0,C 180,E1 -20006.602,E2 -20006.602} C_VEL
LIN {X 0,Y 227.903,Z 429.596,A -85,B 0,C 180,E1 -20010.295,E2 -20010.295} C_VEL
LIN {X 0,Y 227.885,Z 429.599,A -85,B 0,C 180,E1 -20013.718,E2 -20013.718} C_VEL
LIN {X 0,Y 227.866,Z 429.601,A -85,B 0,C 180,E1 -20018.085,E2 -20018.085} C_VEL
LIN {X 0,Y 227.926,Z 429.591,A -85,B 0,C 180,E1 -20022.714,E2 -20022.714} C_VEL
LIN {X 0,Y 227.929,Z 429.593,A -85,B 0,C 180,E1 -20027.286,E2 -20027.286} C_VEL
LIN {X 0,Y 227.867,Z 429.602,A -85,B 0,C 180,E1 -20031.915,E2 -20031.915} C_VEL
LIN {X 0,Y 227.886,Z 429.599,A -85,B 0,C 180,E1 -20036.373,E2 -20036.373} C_VEL
LIN {X 0,Y 227.905,Z 429.597,A -85,B 0,C 180,E1 -20036.847,E2 -20036.847} C_VEL
LIN {X 0,Y 229.022,Z 432.627,A -85,B 0,C 180,E1 -20037.204,E2 -20037.204} C_VEL
LIN {X 0,Y 230.327,Z 434.937,A -85,B 0,C 180,E1 -20037.528,E2 -20037.528} C_VEL
LIN {X 0,Y 234.982,Z 443.832,A -85,B 0,C 180,E1 -20038.78,E2 -20038.78} C_VEL
LIN {X 0,Y 239.118,Z 452.908,A -85,B 0,C 180,E1 -20040.113,E2 -20040.113} C_VEL
LIN {X 0,Y 242.806,Z 462.954,A -85,B 0,C 180,E1 -20041.656,E2 -20041.656} C_VEL
LIN {X 0,Y 246.738,Z 472.229,A -85,B 0,C 180,E1 -20043.334,E2 -20043.334} C_VEL
LIN {X 0,Y 251.642,Z 481.045,A -85,B 0,C 180,E1 -20045.234,E2 -20045.234} C_VEL
LIN {X 0,Y 257.562,Z 489.419,A -85,B 0,C 180,E1 -20047.32,E2 -20047.32} C_VEL
LIN {X 0,Y 265.317,Z 498.418,A -85,B 0,C 180,E1 -20049.858,E2 -20049.858} C_VEL
LIN {X 0,Y 274.284,Z 507.149,A -85,B 0,C 180,E1 -20052.639,E2 -20052.639} C_VEL
LIN {X 0,Y 283.254,Z 514.799,A -85,B 0,C 180,E1 -20055.384,E2 -20055.384} C_VEL
LIN {X 0,Y 289.551,Z 519.804,A -85,B 0,C 180,E1 -20057.383,E2 -20057.383} C_VEL
LIN {X 0,Y 294.264,Z 523.403,A -85,B 0,C 180,E1 -20058.985,E2 -20058.985} C_VEL
LIN {X 0,Y 300.492,Z 528.114,A -85,B 0,C 180,E1 -20061.392,E2 -20061.392} C_VEL
LIN {X 0,Y 303.273,Z 530.239,A -85,B 0,C 180,E1 -20062.678,E2 -20062.678} C_VEL
LIN {X 0,Y 306.563,Z 533.018,A -85,B 0,C 180,E1 -20064.739,E2 -20064.739} C_VEL
LIN {X 0,Y 309.657,Z 534.947,A -85,B 0,C 180,E1 -20066.981,E2 -20066.981} C_VEL
LIN {X 0,Y 311.364,Z 535.674,A -85,B 0,C 180,E1 -20068.707,E2 -20068.707} C_VEL
LIN {X 0,Y 311.992,Z 535.828,A -85,B 0,C 180,E1 -20070,E2 -20070} C_VEL
LIN {X 0,Y 311.362,Z 535.673,A -85,B 0,C 180,E1 -20071.294,E2 -20071.294} C_VEL
LIN {X 0,Y 309.656,Z 534.95,A -85,B 0,C 180,E1 -20073.015,E2 -20073.015} C_VEL
LIN {X 0,Y 306.545,Z 533.018,A -85,B 0,C 180,E1 -20075.262,E2 -20075.262} C_VEL
LIN {X 0,Y 303.247,Z 530.239,A -85,B 0,C 180,E1 -20077.323,E2 -20077.323} C_VEL
LIN {X 0,Y 300.452,Z 528.118,A -85,B 0,C 180,E1 -20078.608,E2 -20078.608} C_VEL
LIN {X 0,Y 296.372,Z 525.031,A -85,B 0,C 180,E1 -20080.245,E2 -20080.245} C_VEL
LIN {X 0,Y 291.991,Z 521.652,A -85,B 0,C 180,E1 -20081.805,E2 -20081.805} C_VEL
LIN {X 0,Y 285.881,Z 516.813,A -85,B 0,C 180,E1 -20083.826,E2 -20083.826} C_VEL
LIN {X 0,Y 276.912,Z 509.475,A -85,B 0,C 180,E1 -20086.557,E2 -20086.557} C_VEL
LIN {X 0,Y 268.056,Z 501.204,A -85,B 0,C 180,E1 -20089.293,E2 -20089.293} C_VEL
LIN {X 0,Y 259.59,Z 491.962,A -85,B 0,C 180,E1 -20091.992,E2 -20091.992} C_VEL
LIN {X 0,Y 252.7,Z 482.682,A -85,B 0,C 180,E1 -20094.382,E2 -20094.382} C_VEL
LIN {X 0,Y 247.259,Z 473.302,A -85,B 0,C 180,E1 -20096.452,E2 -20096.452} C_VEL
LIN {X 0,Y 243.477,Z 464.711,A -85,B 0,C 180,E1 -20098.05,E2 -20098.05} C_VEL
LIN {X 0,Y 239.541,Z 454.057,A -85,B 0,C 180,E1 -20099.719,E2 -20099.719} C_VEL
LIN {X 0,Y 235.722,Z 445.347,A -85,B 0,C 180,E1 -20101.001,E2 -20101.001} C_VEL
LIN {X 0,Y 230.997,Z 436.101,A -85,B 0,C 180,E1 -20102.326,E2 -20102.326} C_VEL
LIN {X 0,Y 228.849,Z 432.311,A -85,B 0,C 180,E1 -20102.851,E2 -20102.851} C_VEL
LIN {X 0,Y 227.903,Z 429.597,A -85,B 0,C 180,E1 -20103.152,E2 -20103.152} C_VEL
LIN {X 0,Y 227.906,Z 429.597,A -85,B 0,C 180,E1 -20106.702,E2 -20106.702} C_VEL
LIN {X 0,Y 227.889,Z 429.598,A -85,B 0,C 180,E1 -20110.363,E2 -20110.363} C_VEL
LIN {X 0,Y 227.906,Z 429.596,A -85,B 0,C 180,E1 -20112.72,E2 -20112.72} C_VEL
LIN {X 0,Y 227.845,Z 429.602,A -85,B 0,C 180,E1 -20117.756,E2 -20117.756} C_VEL
LIN {X 0,Y 227.867,Z 429.6,A -85,B 0,C 180,E1 -20121.915,E2 -20121.915} C_VEL
LIN {X 0,Y 227.888,Z 429.598,A -85,B 0,C 180,E1 -20126.374,E2 -20126.374} C_VEL
LIN {X 0,Y 227.916,Z 429.594,A -85,B 0,C 180,E1 -20130.439,E2 -20130.439} C_VEL
LIN {X 0,Y 227.926,Z 429.587,A -85,B 0,C 180,E1 -20134.427,E2 -20134.427} C_VEL
LIN {X 0,Y 227.96,Z 429.588,A -85,B 0,C 180,E1 -20138.288,E2 -20138.288} C_VEL
LIN {X 0,Y 228.033,Z 429.579,A -85,B 0,C 180,E1 -20142.827,E2 -20142.827} C_VEL
LIN {X 0,Y 228.092,Z 429.573,A -85,B 0,C 180,E1 -20147.545,E2 -20147.545} C_VEL
LIN {X 0,Y 228.304,Z 429.542,A -85,B 0,C 180,E1 -20151.147,E2 -20151.147} C_VEL
LIN {X 0,Y 228.354,Z 429.539,A -85,B 0,C 180,E1 -20152.93,E2 -20152.93} C_VEL
LIN {X 0,Y 228.553,Z 429.491,A -85,B 0,C 180,E1 -20158.239,E2 -20158.239} C_VEL
LIN {X 0,Y 228.554,Z 429.513,A -85,B 0,C 180,E1 -20161.763,E2 -20161.763} C_VEL
LIN {X 0,Y 228.357,Z 429.539,A -85,B 0,C 180,E1 -20167.072,E2 -20167.072} C_VEL
LIN {X 0,Y 228.167,Z 429.563,A -85,B 0,C 180,E1 -20170.651,E2 -20170.651} C_VEL
LIN {X 0,Y 228.065,Z 429.576,A -85,B 0,C 180,E1 -20174.273,E2 -20174.273} C_VEL
LIN {X 0,Y 228.004,Z 429.584,A -85,B 0,C 180,E1 -20177.954,E2 -20177.954} C_VEL
LIN {X 0,Y 227.931,Z 429.592,A -85,B 0,C 180,E1 -20182.33,E2 -20182.33} C_VEL
LIN {X 0,Y 227.943,Z 429.591,A -85,B 0,C 180,E1 -20186.603,E2 -20186.603} C_VEL
LIN {X 0,Y 227.885,Z 429.599,A -85,B 0,C 180,E1 -20187.556,E2 -20187.556} C_VEL
LIN {X 0,Y 228.116,Z 431.2,A -85,B 0,C 180,E1 -20191.585,E2 -20191.585} C_VEL
LIN {X 0,Y 228.366,Z 433.161,A -85,B 0,C 180,E1 -20195.785,E2 -20195.785} C_VEL
LIN {X 0,Y 228.7,Z 435.453,A -85,B 0,C 180,E1 -20200.192,E2 -20200.192} C_VEL
LIN {X 0,Y 228.904,Z 436.785,A -85,B 0,C 180,E1 -20202.535,E2 -20202.535} C_VEL
LIN {X 0,Y 229.022,Z 438.325,A -85,B 0,C 180,E1 -20205.106,E2 -20205.106} C_VEL
LIN {X 0,Y 229.006,Z 439.85,A -85,B 0,C 180,E1 -20207.534,E2 -20207.534} C_VEL
LIN {X 0,Y 228.72,Z 441.627,A -85,B 0,C 180,E1 -20210.193,E2 -20210.193} C_VEL
LIN {X 0,Y 228.026,Z 444.441,A -85,B 0,C 180,E1 -20214.155,E2 -20214.155} C_VEL
LIN {X 0,Y 227.552,Z 446.608,A -85,B 0,C 180,E1 -20217.08,E2 -20217.08} C_VEL
LIN {X 0,Y 228.349,Z 449.684,A -85,B 0,C 180,E1 -20217.371,E2 -20217.371} C_VEL
LIN {X 0,Y 232.392,Z 462.797,A -85,B 0,C 180,E1 -20218.948,E2 -20218.948} C_VEL
LIN {X 0,Y 234.9,Z 473.966,A -85,B 0,C 180,E1 -20220.447,E2 -20220.447} C_VEL
LIN {X 0,Y 236.458,Z 484.654,A -85,B 0,C 180,E1 -20222.037,E2 -20222.037} C_VEL
LIN {X 0,Y 237.128,Z 492.931,A -85,B 0,C 180,E1 -20223.405,E2 -20223.405} C_VEL
LIN {X 0,Y 237.293,Z 500.377,A -85,B 0,C 180,E1 -20224.759,E2 -20224.759} C_VEL
LIN {X 0,Y 236.425,Z 503.496,A -85,B 0,C 180,E1 -20225.304,E2 -20225.304} C_VEL
LIN {X 0,Y 233.695,Z 507.553,A -85,B 0,C 180,E1 -20225.873,E2 -20225.873} C_VEL
LIN {X 0,Y 228.946,Z 513.187,A -85,B 0,C 180,E1 -20226.754,E2 -20226.754} C_VEL
LIN {X 0,Y 227.499,Z 516.002,A -85,B 0,C 180,E1 -20227.387,E2 -20227.387} C_VEL
LIN {X 0,Y 225.549,Z 523.754,A -85,B 0,C 180,E1 -20229.57,E2 -20229.57} C_VEL
LIN {X 0,Y 223.609,Z 530.026,A -85,B 0,C 180,E1 -20231.681,E2 -20231.681} C_VEL
LIN {X 0,Y 222.336,Z 534.531,A -85,B 0,C 180,E1 -20233.472,E2 -20233.472} C_VEL
LIN {X 0,Y 220.722,Z 540.025,A -85,B 0,C 180,E1 -20236.184,E2 -20236.184} C_VEL
LIN {X 0,Y 219.667,Z 544.357,A -85,B 0,C 180,E1 -20238.932,E2 -20238.932} C_VEL
LIN {X 0,Y 219.146,Z 546.729,A -85,B 0,C 180,E1 -20240.773,E2 -20240.773} C_VEL
LIN {X 0,Y 218.799,Z 548.533,A -85,B 0,C 180,E1 -20242.618,E2 -20242.618} C_VEL
LIN {X 0,Y 218.516,Z 550.989,A -85,B 0,C 180,E1 -20246.312,E2 -20246.312} C_VEL
LIN {X 0,Y 218.561,Z 551.584,A -85,B 0,C 180,E1 -20248.157,E2 -20248.157} C_VEL
LIN {X 0,Y 218.61,Z 551.741,A -85,B 0,C 180,E1 -20250,E2 -20250} C_VEL
LIN {X 0,Y 218.562,Z 551.584,A -85,B 0,C 180,E1 -20251.842,E2 -20251.842} C_VEL
LIN {X 0,Y 218.555,Z 550.57,A -85,B 0,C 180,E1 -20254.535,E2 -20254.535} C_VEL
LIN {X 0,Y 218.8,Z 548.533,A -85,B 0,C 180,E1 -20257.381,E2 -20257.381} C_VEL
LIN {X 0,Y 219.375,Z 545.577,A -85,B 0,C 180,E1 -20260.148,E2 -20260.148} C_VEL
LIN {X 0,Y 220.326,Z 541.582,A -85,B 0,C 180,E1 -20262.902,E2 -20262.902} C_VEL
LIN {X 0,Y 221.741,Z 536.449,A -85,B 0,C 180,E1 -20265.628,E2 -20265.628} C_VEL
LIN {X 0,Y 223.297,Z 531.185,A -85,B 0,C 180,E1 -20267.87,E2 -20267.87} C_VEL
LIN {X 0,Y 225.174,Z 524.868,A -85,B 0,C 180,E1 -20270.079,E2 -20270.079} C_VEL
LIN {X 0,Y 226.719,Z 518.911,A -85,B 0,C 180,E1 -20271.837,E2 -20271.837} C_VEL
LIN {X 0,Y 228.576,Z 511.983,A -85,B 0,C 180,E1 -20273.559,E2 -20273.559} C_VEL
LIN {X 0,Y 230.605,Z 503.802,A -85,B 0,C 180,E1 -20275.256,E2 -20275.256} C_VEL
LIN {X 0,Y 230.564,Z 495.224,A -85,B 0,C 180,E1 -20276.962,E2 -20276.962} C_VEL
LIN {X 0,Y 230.15,Z 488.08,A -85,B 0,C 180,E1 -20278.248,E2 -20278.248} C_VEL
LIN {X 0,Y 228.953,Z 478.374,A -85,B 0,C 180,E1 -20279.822,E2 -20279.822} C_VEL
LIN {X 0,Y 227.099,Z 468.671,A -85,B 0,C 180,E1 -20281.25,E2 -20281.25} C_VEL
LIN {X 0,Y 224.086,Z 457.315,A -85,B 0,C 180,E1 -20282.772,E2 -20282.772} C_VEL
LIN {X 0,Y 221.396,Z 449.437,A -85,B 0,C 180,E1 -20283.789,E2 -20283.789} C_VEL
LIN {X 0,Y 220.61,Z 446.387,A -85,B 0,C 180,E1 -20284.123,E2 -20284.123} C_VEL
LIN {X 0,Y 221.217,Z 444.023,A -85,B 0,C 180,E1 -20287.415,E2 -20287.415} C_VEL
LIN {X 0,Y 221.84,Z 441.151,A -85,B 0,C 180,E1 -20291.703,E2 -20291.703} C_VEL
LIN {X 0,Y 221.928,Z 439.622,A -85,B 0,C 180,E1 -20294.161,E2 -20294.161} C_VEL
LIN {X 0,Y 221.746,Z 437.251,A -85,B 0,C 180,E1 -20298.273,E2 -20298.273} C_VEL
LIN {X 0,Y 221.392,Z 434.832,A -85,B 0,C 180,E1 -20302.903,E2 -20302.903} C_VEL
LIN {X 0,Y 221.14,Z 432.771,A -85,B 0,C 180,E1 -20307.297,E2 -20307.297} C_VEL
LIN {X 0,Y 220.912,Z 431.024,A -85,B 0,C 180,E1 -20311.496,E2 -20311.496} C_VEL
LIN {X 0,Y 220.894,Z 430.474,A -85,B 0,C 180,E1 -20313.548,E2 -20313.548} C_VEL
LIN {X 0,Y 220.876,Z 430.477,A -85,B 0,C 180,E1 -20317.552,E2 -20317.552} C_VEL
LIN {X 0,Y 220.982,Z 430.461,A -85,B 0,C 180,E1 -20322.57,E2 -20322.57} C_VEL
LIN {X 0,Y 221.01,Z 430.455,A -85,B 0,C 180,E1 -20327.137,E2 -20327.137} C_VEL
LIN {X 0,Y 221.255,Z 430.425,A -85,B 0,C 180,E1 -20330.861,E2 -20330.861} C_VEL
LIN {X 0,Y 221.308,Z 430.419,A -85,B 0,C 180,E1 -20332.701,E2 -20332.701} C_VEL
LIN {X 0,Y 221.509,Z 430.391,A -85,B 0,C 180,E1 -20338.181,E2 -20338.181} C_VEL
LIN {X 0,Y 221.508,Z 430.367,A -85,B 0,C 180,E1 -20341.817,E2 -20341.817} C_VEL
LIN {X 0,Y 221.286,Z 430.42,A -85,B 0,C 180,E1 -20347.298,E2 -20347.298} C_VEL
LIN {X 0,Y 221.108,Z 430.441,A -85,B 0,C 180,E1 -20350.993,E2 -20350.993} C_VEL
LIN {X 0,Y 221.012,Z 430.455,A -85,B 0,C 180,E1 -20356.629,E2 -20356.629} C_VEL
LIN {X 0,Y 220.888,Z 430.466,A -85,B 0,C 180,E1 -20360.485,E2 -20360.485} C_VEL
LIN {X 0,Y 220.862,Z 430.467,A -85,B 0,C 180,E1 -20364.434,E2 -20364.434} C_VEL
LIN {X 0,Y 220.831,Z 430.476,A -85,B 0,C 180,E1 -20368.513,E2 -20368.513} C_VEL
LIN {X 0,Y 220.819,Z 430.478,A -85,B 0,C 180,E1 -20372.754,E2 -20372.754} C_VEL
LIN {X 0,Y 220.833,Z 430.477,A -85,B 0,C 180,E1 -20377.288,E2 -20377.288} C_VEL
LIN {X 0,Y 220.866,Z 430.473,A -85,B 0,C 180,E1 -20381.929,E2 -20381.929} C_VEL
LIN {X 0,Y 220.87,Z 430.472,A -85,B 0,C 180,E1 -20385.572,E2 -20385.572} C_VEL
LIN {X 0,Y 220.856,Z 430.474,A -85,B 0,C 180,E1 -20389.791,E2 -20389.791} C_VEL
LIN {X 0,Y 220.83,Z 430.478,A -85,B 0,C 180,E1 -20392.795,E2 -20392.795} C_VEL
LIN {X 0,Y 220.818,Z 430.481,A -85,B 0,C 180,E1 -20395.682,E2 -20395.682} C_VEL
LIN {X 0,Y 221.854,Z 433.369,A -85,B 0,C 180,E1 -20396.028,E2 -20396.028} C_VEL
LIN {X 0,Y 223.218,Z 435.496,A -85,B 0,C 180,E1 -20396.375,E2 -20396.375} C_VEL
LIN {X 0,Y 228.43,Z 445.528,A -85,B 0,C 180,E1 -20397.889,E2 -20397.889} C_VEL
LIN {X 0,Y 232.719,Z 455.012,A -85,B 0,C 180,E1 -20399.39,E2 -20399.39} C_VEL
LIN {X 0,Y 236.285,Z 464.836,A -85,B 0,C 180,E1 -20401.003,E2 -20401.003} C_VEL
LIN {X 0,Y 239.783,Z 473.787,A -85,B 0,C 180,E1 -20402.692,E2 -20402.692} C_VEL
LIN {X 0,Y 244.651,Z 483.19,A -85,B 0,C 180,E1 -20404.804,E2 -20404.804} C_VEL
LIN {X 0,Y 249.761,Z 490.839,A -85,B 0,C 180,E1 -20406.801,E2 -20406.801} C_VEL
LIN {X 0,Y 257.137,Z 499.614,A -85,B 0,C 180,E1 -20409.403,E2 -20409.403} C_VEL
LIN {X 0,Y 265.673,Z 508.094,A -85,B 0,C 180,E1 -20412.234,E2 -20412.234} C_VEL
LIN {X 0,Y 275.019,Z 515.849,A -85,B 0,C 180,E1 -20415.195,E2 -20415.195} C_VEL
LIN {X 0,Y 281.135,Z 520.451,A -85,B 0,C 180,E1 -20417.144,E2 -20417.144} C_VEL
LIN {X 0,Y 288.228,Z 525.565,A -85,B 0,C 180,E1 -20419.597,E2 -20419.597} C_VEL
LIN {X 0,Y 293.706,Z 529.368,A -85,B 0,C 180,E1 -20421.746,E2 -20421.746} C_VEL
LIN {X 0,Y 296.804,Z 531.515,A -85,B 0,C 180,E1 -20423.201,E2 -20423.201} C_VEL
LIN {X 0,Y 299.003,Z 533.245,A -85,B 0,C 180,E1 -20424.606,E2 -20424.606} C_VEL
LIN {X 0,Y 300.989,Z 534.57,A -85,B 0,C 180,E1 -20425.984,E2 -20425.984} C_VEL
LIN {X 0,Y 302.835,Z 535.506,A -85,B 0,C 180,E1 -20427.34,E2 -20427.34} C_VEL
LIN {X 0,Y 304.156,Z 536.063,A -85,B 0,C 180,E1 -20428.676,E2 -20428.676} C_VEL
LIN {X 0,Y 304.888,Z 536.245,A -85,B 0,C 180,E1 -20430,E2 -20430} C_VEL
LIN {X 0,Y 304.153,Z 536.063,A -85,B 0,C 180,E1 -20431.324,E2 -20431.324} C_VEL
LIN {X 0,Y 302.574,Z 535.389,A -85,B 0,C 180,E1 -20432.854,E2 -20432.854} C_VEL
LIN {X 0,Y 300.981,Z 534.569,A -85,B 0,C 180,E1 -20434.017,E2 -20434.017} C_VEL
LIN {X 0,Y 298.972,Z 533.245,A -85,B 0,C 180,E1 -20435.396,E2 -20435.396} C_VEL
LIN {X 0,Y 296.763,Z 531.516,A -85,B 0,C 180,E1 -20436.801,E2 -20436.801} C_VEL
LIN {X 0,Y 293.647,Z 529.369,A -85,B 0,C 180,E1 -20438.256,E2 -20438.256} C_VEL
LIN {X 0,Y 288.253,Z 525.56,A -85,B 0,C 180,E1 -20440.404,E2 -20440.404} C_VEL
LIN {X 0,Y 280.698,Z 520.072,A -85,B 0,C 180,E1 -20443.023,E2 -20443.023} C_VEL
LIN {X 0,Y 272.317,Z 513.689,A -85,B 0,C 180,E1 -20445.668,E2 -20445.668} C_VEL
LIN {X 0,Y 262.755,Z 505.317,A -85,B 0,C 180,E1 -20448.722,E2 -20448.722} C_VEL
LIN {X 0,Y 254.161,Z 496.313,A -85,B 0,C 180,E1 -20451.618,E2 -20451.618} C_VEL
LIN {X 0,Y 247.419,Z 487.487,A -85,B 0,C 180,E1 -20454.104,E2 -20454.104} C_VEL
LIN {X 0,Y 241.807,Z 478.067,A -85,B 0,C 180,E1 -20456.403,E2 -20456.403} C_VEL
LIN {X 0,Y 237.34,Z 467.805,A -85,B 0,C 180,E1 -20458.483,E2 -20458.483} C_VEL
LIN {X 0,Y 233.248,Z 456.306,A -85,B 0,C 180,E1 -20460.405,E2 -20460.405} C_VEL
LIN {X 0,Y 228.867,Z 446.422,A -85,B 0,C 180,E1 -20461.975,E2 -20461.975} C_VEL
LIN {X 0,Y 223.606,Z 436.263,A -85,B 0,C 180,E1 -20463.538,E2 -20463.538} C_VEL
LIN {X 0,Y 222.145,Z 433.757,A -85,B 0,C 180,E1 -20463.919,E2 -20463.919} C_VEL
LIN {X 0,Y 221.002,Z 431.417,A -85,B 0,C 180,E1 -20464.229,E2 -20464.229} C_VEL
LIN {X 0,Y 220.82,Z 430.48,A -85,B 0,C 180,E1 -20464.318,E2 -20464.318} C_VEL
LIN {X 0,Y 220.835,Z 430.477,A -85,B 0,C 180,E1 -20467.288,E2 -20467.288} C_VEL
LIN {X 0,Y 220.85,Z 430.476,A -85,B 0,C 180,E1 -20471.934,E2 -20471.934} C_VEL
LIN {X 0,Y 220.808,Z 430.479,A -85,B 0,C 180,E1 -20475.556,E2 -20475.556} C_VEL
LIN {X 0,Y 220.807,Z 430.481,A -85,B 0,C 180,E1 -20480.465,E2 -20480.465} C_VEL
LIN {X 0,Y 220.829,Z 430.477,A -85,B 0,C 180,E1 -20482.795,E2 -20482.795} C_VEL
LIN {X 0,Y 220.822,Z 430.477,A -85,B 0,C 180,E1 -20487.246,E2 -20487.246} C_VEL
LIN {X 0,Y 220.834,Z 430.476,A -85,B 0,C 180,E1 -20491.487,E2 -20491.487} C_VEL
LIN {X 0,Y 220.865,Z 430.466,A -85,B 0,C 180,E1 -20495.566,E2 -20495.566} C_VEL
LIN {X 0,Y 220.89,Z 430.465,A -85,B 0,C 180,E1 -20499.515,E2 -20499.515} C_VEL
LIN {X 0,Y 221.015,Z 430.454,A -85,B 0,C 180,E1 -20503.371,E2 -20503.371} C_VEL
LIN {X 0,Y 221.111,Z 430.44,A -85,B 0,C 180,E1 -20509.007,E2 -20509.007} C_VEL
LIN {X 0,Y 221.289,Z 430.419,A -85,B 0,C 180,E1 -20512.703,E2 -20512.703} C_VEL
LIN {X 0,Y 221.511,Z 430.366,A -85,B 0,C 180,E1 -20518.183,E2 -20518.183} C_VEL
LIN {X 0,Y 221.512,Z 430.391,A -85,B 0,C 180,E1 -20521.819,E2 -20521.819} C_VEL
LIN {X 0,Y 221.311,Z 430.418,A -85,B 0,C 180,E1 -20527.299,E2 -20527.299} C_VEL
LIN {X 0,Y 221.111,Z 430.443,A -85,B 0,C 180,E1 -20530.995,E2 -20530.995} C_VEL
LIN {X 0,Y 221.017,Z 430.454,A -85,B 0,C 180,E1 -20536.631,E2 -20536.631} C_VEL
LIN {X 0,Y 220.893,Z 430.47,A -85,B 0,C 180,E1 -20540.487,E2 -20540.487} C_VEL
LIN {X 0,Y 220.868,Z 430.473,A -85,B 0,C 180,E1 -20544.436,E2 -20544.436} C_VEL
LIN {X 0,Y 220.886,Z 430.472,A -85,B 0,C 180,E1 -20547.016,E2 -20547.016} C_VEL
LIN {X 0,Y 221.073,Z 431.978,A -85,B 0,C 180,E1 -20550.87,E2 -20550.87} C_VEL
LIN {X 0,Y 221.27,Z 433.77,A -85,B 0,C 180,E1 -20554.871,E2 -20554.871} C_VEL
LIN {X 0,Y 221.585,Z 435.992,A -85,B 0,C 180,E1 -20559.372,E2 -20559.372} C_VEL
LIN {X 0,Y 221.853,Z 438.107,A -85,B 0,C 180,E1 -20563.231,E2 -20563.231} C_VEL
LIN {X 0,Y 221.933,Z 440.189,A -85,B 0,C 180,E1 -20566.749,E2 -20566.749} C_VEL
LIN {X 0,Y 221.552,Z 442.695,A -85,B 0,C 180,E1 -20570.622,E2 -20570.622} C_VEL
LIN {X 0,Y 221.21,Z 444.224,A -85,B 0,C 180,E1 -20572.869,E2 -20572.869} C_VEL
LIN {X 0,Y 220.618,Z 446.423,A -85,B 0,C 180,E1 -20575.922,E2 -20575.922} C_VEL
LIN {X 0,Y 221.505,Z 449.632,A -85,B 0,C 180,E1 -20576.24,E2 -20576.24} C_VEL
LIN {X 0,Y 224.874,Z 459.877,A -85,B 0,C 180,E1 -20577.549,E2 -20577.549} C_VEL
LIN {X 0,Y 227.917,Z 472.308,A -85,B 0,C 180,E1 -20579.267,E2 -20579.267} C_VEL
LIN {X 0,Y 229.616,Z 483.286,A -85,B 0,C 180,E1 -20580.954,E2 -20580.954} C_VEL
LIN {X 0,Y 230.475,Z 492.709,A -85,B 0,C 180,E1 -20582.574,E2 -20582.574} C_VEL
LIN {X 0,Y 230.598,Z 501.831,A -85,B 0,C 180,E1 -20584.327,E2 -20584.327} C_VEL
LIN {X 0,Y 230.175,Z 506.071,A -85,B 0,C 180,E1 -20585.176,E2 -20585.176} C_VEL
LIN {X 0,Y 227.499,Z 516.002,A -85,B 0,C 180,E1 -20587.387,E2 -20587.387} C_VEL
LIN {X 0,Y 225.778,Z 520.096,A -85,B 0,C 180,E1 -20588.409,E2 -20588.409} C_VEL
LIN {X 0,Y 221.349,Z 526.16,A -85,B 0,C 180,E1 -20590.046,E2 -20590.046} C_VEL
LIN {X 0,Y 216.98,Z 531.743,A -85,B 0,C 180,E1 -20591.858,E2 -20591.858} C_VEL
LIN {X 0,Y 215.381,Z 534.744,A -85,B 0,C 180,E1 -20593.138,E2 -20593.138} C_VEL
LIN {X 0,Y 213.797,Z 539.812,A -85,B 0,C 180,E1 -20595.727,E2 -20595.727} C_VEL
LIN {X 0,Y 212.688,Z 544.146,A -85,B 0,C 180,E1 -20598.564,E2 -20598.564} C_VEL
LIN {X 0,Y 212.113,Z 546.516,A -85,B 0,C 180,E1 -20600.464,E2 -20600.464} C_VEL
LIN {X 0,Y 211.728,Z 548.32,A -85,B 0,C 180,E1 -20602.37,E2 -20602.37} C_VEL
LIN {X 0,Y 211.44,Z 550.778,A -85,B 0,C 180,E1 -20606.188,E2 -20606.188} C_VEL
LIN {X 0,Y 211.461,Z 551.372,A -85,B 0,C 180,E1 -20608.095,E2 -20608.095} C_VEL
LIN {X 0,Y 211.528,Z 551.53,A -85,B 0,C 180,E1 -20610,E2 -20610} C_VEL
LIN {X 0,Y 211.462,Z 551.372,A -85,B 0,C 180,E1 -20611.904,E2 -20611.904} C_VEL
LIN {X 0,Y 211.476,Z 550.516,A -85,B 0,C 180,E1 -20614.434,E2 -20614.434} C_VEL
LIN {X 0,Y 211.73,Z 548.321,A -85,B 0,C 180,E1 -20617.629,E2 -20617.629} C_VEL
LIN {X 0,Y 212.377,Z 545.365,A -85,B 0,C 180,E1 -20620.486,E2 -20620.486} C_VEL
LIN {X 0,Y 213.362,Z 541.37,A -85,B 0,C 180,E1 -20623.33,E2 -20623.33} C_VEL
LIN {X 0,Y 214.896,Z 536.237,A -85,B 0,C 180,E1 -20626.139,E2 -20626.139} C_VEL
LIN {X 0,Y 216.49,Z 530.972,A -85,B 0,C 180,E1 -20628.452,E2 -20628.452} C_VEL
LIN {X 0,Y 218.491,Z 524.656,A -85,B 0,C 180,E1 -20630.721,E2 -20630.721} C_VEL
LIN {X 0,Y 220.109,Z 518.699,A -85,B 0,C 180,E1 -20632.528,E2 -20632.528} C_VEL
LIN {X 0,Y 222.058,Z 511.771,A -85,B 0,C 180,E1 -20634.295,E2 -20634.295} C_VEL
LIN {X 0,Y 223.905,Z 504.725,A -85,B 0,C 180,E1 -20635.817,E2 -20635.817} C_VEL
LIN {X 0,Y 223.958,Z 496.364,A -85,B 0,C 180,E1 -20637.571,E2 -20637.571} C_VEL
LIN {X 0,Y 223.449,Z 487.854,A -85,B 0,C 180,E1 -20639.175,E2 -20639.175} C_VEL
LIN {X 0,Y 222.186,Z 477.534,A -85,B 0,C 180,E1 -20640.906,E2 -20640.906} C_VEL
LIN {X 0,Y 220.375,Z 468.447,A -85,B 0,C 180,E1 -20642.316,E2 -20642.316} C_VEL
LIN {X 0,Y 217.281,Z 457.005,A -85,B 0,C 180,E1 -20643.941,E2 -20643.941} C_VEL
LIN {X 0,Y 214.626,Z 449.443,A -85,B 0,C 180,E1 -20644.993,E2 -20644.993} C_VEL
LIN {X 0,Y 213.737,Z 446.201,A -85,B 0,C 180,E1 -20645.343,E2 -20645.343} C_VEL
LIN {X 0,Y 214.319,Z 444.001,A -85,B 0,C 180,E1 -20648.538,E2 -20648.538} C_VEL
LIN {X 0,Y 214.713,Z 442.289,A -85,B 0,C 180,E1 -20651.162,E2 -20651.162} C_VEL
LIN {X 0,Y 214.9,Z 440.586,A -85,B 0,C 180,E1 -20653.987,E2 -20653.987} C_VEL
LIN {X 0,Y 214.812,Z 439.09,A -85,B 0,C 180,E1 -20656.601,E2 -20656.601} C_VEL
LIN {X 0,Y 214.655,Z 437.744,A -85,B 0,C 180,E1 -20659.093,E2 -20659.093} C_VEL
LIN {X 0,Y 214.291,Z 435.404,A -85,B 0,C 180,E1 -20663.818,E2 -20663.818} C_VEL
LIN {X 0,Y 214.051,Z 433.278,A -85,B 0,C 180,E1 -20668.61,E2 -20668.61} C_VEL
LIN {X 0,Y 213.864,Z 431.717,A -85,B 0,C 180,E1 -20672.607,E2 -20672.607} C_VEL
LIN {X 0,Y 213.846,Z 431.354,A -85,B 0,C 180,E1 -20676.772,E2 -20676.772} C_VEL
LIN {X 0,Y 213.941,Z 431.338,A -85,B 0,C 180,E1 -20682.802,E2 -20682.802} C_VEL
LIN {X 0,Y 213.951,Z 431.336,A -85,B 0,C 180,E1 -20686.705,E2 -20686.705} C_VEL
LIN {X 0,Y 214.194,Z 431.306,A -85,B 0,C 180,E1 -20690.556,E2 -20690.556} C_VEL
LIN {X 0,Y 214.245,Z 431.299,A -85,B 0,C 180,E1 -20692.459,E2 -20692.459} C_VEL
LIN {X 0,Y 214.442,Z 431.272,A -85,B 0,C 180,E1 -20698.121,E2 -20698.121} C_VEL
LIN {X 0,Y 214.546,Z 431.244,A -85,B 0,C 180,E1 -20699.999,E2 -20699.999} C_VEL
LIN {X 0,Y 214.442,Z 431.245,A -85,B 0,C 180,E1 -20701.877,E2 -20701.877} C_VEL
LIN {X 0,Y 214.223,Z 431.3,A -85,B 0,C 180,E1 -20707.539,E2 -20707.539} C_VEL
LIN {X 0,Y 214.04,Z 431.321,A -85,B 0,C 180,E1 -20711.361,E2 -20711.361} C_VEL
LIN {X 0,Y 213.928,Z 431.33,A -85,B 0,C 180,E1 -20715.236,E2 -20715.236} C_VEL
LIN {X 0,Y 213.835,Z 431.345,A -85,B 0,C 180,E1 -20719.187,E2 -20719.187} C_VEL
LIN {X 0,Y 213.842,Z 431.347,A -85,B 0,C 180,E1 -20723.226,E2 -20723.226} C_VEL
LIN {X 0,Y 213.824,Z 431.35,A -85,B 0,C 180,E1 -20727.449,E2 -20727.449} C_VEL
LIN {X 0,Y 213.774,Z 431.356,A -85,B 0,C 180,E1 -20731.735,E2 -20731.735} C_VEL
LIN {X 0,Y 213.75,Z 431.36,A -85,B 0,C 180,E1 -20736.286,E2 -20736.286} C_VEL
LIN {X 0,Y 213.818,Z 431.349,A -85,B 0,C 180,E1 -20741.099,E2 -20741.099} C_VEL
LIN {X 0,Y 213.831,Z 431.35,A -85,B 0,C 180,E1 -20743.693,E2 -20743.693} C_VEL
LIN {X 0,Y 213.836,Z 431.349,A -85,B 0,C 180,E1 -20746.356,E2 -20746.356} C_VEL
LIN {X 0,Y 213.819,Z 431.351,A -85,B 0,C 180,E1 -20749.11,E2 -20749.11} C_VEL
LIN {X 0,Y 213.75,Z 431.361,A -85,B 0,C 180,E1 -20753.714,E2 -20753.714} C_VEL
LIN {X 0,Y 213.742,Z 431.361,A -85,B 0,C 180,E1 -20754.409,E2 -20754.409} C_VEL
LIN {X 0,Y 214.78,Z 434.22,A -85,B 0,C 180,E1 -20754.779,E2 -20754.779} C_VEL
LIN {X 0,Y 216.287,Z 436.621,A -85,B 0,C 180,E1 -20755.192,E2 -20755.192} C_VEL
LIN {X 0,Y 220.494,Z 444.431,A -85,B 0,C 180,E1 -20756.479,E2 -20756.479} C_VEL
LIN {X 0,Y 225.209,Z 454.405,A -85,B 0,C 180,E1 -20758.165,E2 -20758.165} C_VEL
LIN {X 0,Y 228.741,Z 463.409,A -85,B 0,C 180,E1 -20759.738,E2 -20759.738} C_VEL
LIN {X 0,Y 231.913,Z 472.834,A -85,B 0,C 180,E1 -20761.499,E2 -20761.499} C_VEL
LIN {X 0,Y 235.721,Z 481.551,A -85,B 0,C 180,E1 -20763.435,E2 -20763.435} C_VEL
LIN {X 0,Y 240.825,Z 490.435,A -85,B 0,C 180,E1 -20765.746,E2 -20765.746} C_VEL
LIN {X 0,Y 247.368,Z 498.975,A -85,B 0,C 180,E1 -20768.326,E2 -20768.326} C_VEL
LIN {X 0,Y 255.865,Z 507.819,A -85,B 0,C 180,E1 -20771.37,E2 -20771.37} C_VEL
LIN {X 0,Y 263.358,Z 514.276,A -85,B 0,C 180,E1 -20773.88,E2 -20773.88} C_VEL
LIN {X 0,Y 271.447,Z 520.357,A -85,B 0,C 180,E1 -20776.526,E2 -20776.526} C_VEL
LIN {X 0,Y 279.102,Z 525.566,A -85,B 0,C 180,E1 -20779.123,E2 -20779.123} C_VEL
LIN {X 0,Y 285.387,Z 529.615,A -85,B 0,C 180,E1 -20781.503,E2 -20781.503} C_VEL
LIN {X 0,Y 288.963,Z 531.751,A -85,B 0,C 180,E1 -20783.016,E2 -20783.016} C_VEL
LIN {X 0,Y 291.413,Z 533.473,A -85,B 0,C 180,E1 -20784.465,E2 -20784.465} C_VEL
LIN {X 0,Y 293.505,Z 534.791,A -85,B 0,C 180,E1 -20785.881,E2 -20785.881} C_VEL
LIN {X 0,Y 295.493,Z 535.757,A -85,B 0,C 180,E1 -20787.324,E2 -20787.324} C_VEL
LIN {X 0,Y 296.893,Z 536.278,A -85,B 0,C 180,E1 -20788.644,E2 -20788.644} C_VEL
LIN {X 0,Y 297.747,Z 536.453,A -85,B 0,C 180,E1 -20790,E2 -20790} C_VEL
LIN {X 0,Y 296.889,Z 536.278,A -85,B 0,C 180,E1 -20791.357,E2 -20791.357} C_VEL
LIN {X 0,Y 295.419,Z 535.727,A -85,B 0,C 180,E1 -20792.727,E2 -20792.727} C_VEL
LIN {X 0,Y 293.491,Z 534.791,A -85,B 0,C 180,E1 -20794.12,E2 -20794.12} C_VEL
LIN {X 0,Y 289.975,Z 532.425,A -85,B 0,C 180,E1 -20796.443,E2 -20796.443} C_VEL
LIN {X 0,Y 287.218,Z 530.718,A -85,B 0,C 180,E1 -20797.735,E2 -20797.735} C_VEL
LIN {X 0,Y 281.381,Z 526.995,A -85,B 0,C 180,E1 -20800.069,E2 -20800.069} C_VEL
LIN {X 0,Y 274.603,Z 522.436,A -85,B 0,C 180,E1 -20802.461,E2 -20802.461} C_VEL
LIN {X 0,Y 265.745,Z 516.131,A -85,B 0,C 180,E1 -20805.335,E2 -20805.335} C_VEL
LIN {X 0,Y 257.095,Z 508.941,A -85,B 0,C 180,E1 -20808.212,E2 -20808.212} C_VEL
LIN {X 0,Y 248.708,Z 500.533,A -85,B 0,C 180,E1 -20811.173,E2 -20811.173} C_VEL
LIN {X 0,Y 241.952,Z 492.029,A -85,B 0,C 180,E1 -20813.802,E2 -20813.802} C_VEL
LIN {X 0,Y 236.712,Z 483.519,A -85,B 0,C 180,E1 -20816.09,E2 -20816.09} C_VEL
LIN {X 0,Y 232.726,Z 474.907,A -85,B 0,C 180,E1 -20818.073,E2 -20818.073} C_VEL
